// TwinCAT 3 PLC project BE_ObjektH
// ProgramVersion: 3.1.4023.0
// libraries:
//   EfficientIO Communicator, * (EfficientIO)
//   Lynus Energy Basic, * (Lynus AG)
//   Lynus Energy ModbusTCP, * (Lynus AG)
//   Lynus Persistent Data V1, * (Lynus AG)
//   Lynus Standards, * (Lynus AG)
//   Tc2_ModbusSrv, * (Beckhoff Automation GmbH)
//   Tc2_Standard, * (Beckhoff Automation GmbH)
//   Tc2_System, * (Beckhoff Automation GmbH)
//   Tc2_Utilities, * (Beckhoff Automation GmbH)
//   Tc3_IotBase, * (Beckhoff Automation GmbH)
//   Tc3_JsonXml, * (Beckhoff Automation GmbH)
//   Tc3_Module, * (Beckhoff Automation GmbH)
// project tree:
//   / FastTask.TcTTO, MiddleTask.TcTTO, SlowTask.TcTTO (not stored)
//   FB/ FB_ADS_Read.TcPOU, FB_ECS_Keba_P30.TcPOU, FB_Shelly_3EM_not_tested.TcPOU (excluded from build), FB_Shelly_3EM_Helper_not_tested.TcPOU (excluded from build), FB_Shelly_3EM_Helper.TcPOU, FB_Shelly_3EM.TcPOU, F_AdsErrorText.TcPOU
//   POUs/ prgComEffIO.TcPOU, prgCS.TcPOU, prgMain.TcPOU, prgPersistent.TcPOU, prgPV.TcPOU, prgRWEffIO.TcPOU, prgShelly.TcPOU, prgVarEffIO.TcPOU, prg_SystemTime.TcPOU (not stored)
// real-time tasks:
//   TASK FastTask: cycle T#5ms, priority 19, ADS port 350
//   TASK MiddleTask: cycle T#10ms, priority 20, ADS port 351
//   TASK SlowTask: cycle T#20ms, priority 21, ADS port 352

CONFIGURATION BE_ObjektH
    RESOURCE PLC ON TwinCAT3
        TASK FastTask(INTERVAL := T#5ms, PRIORITY := 19);
        TASK MiddleTask(INTERVAL := T#10ms, PRIORITY := 20);
        PROGRAM prgRWEffIO WITH FastTask : prgRWEffIO;
        PROGRAM prgVarEffIO WITH FastTask : prgVarEffIO;
        PROGRAM prg_SystemTime WITH FastTask : prg_SystemTime;
        PROGRAM prgPV WITH MiddleTask : prgPV;
        PROGRAM prgShelly WITH MiddleTask : prgShelly;
        PROGRAM prgCS WITH MiddleTask : prgCS;
        PROGRAM prgPersistent WITH MiddleTask : prgPersistent;
        PROGRAM prgMain WITH MiddleTask : prgMain;
    END_RESOURCE
END_CONFIGURATION

// ---- POUs/prgRWEffIO.TcPOU
PROGRAM prgRWEffIO
VAR
	fbRW1		: FB_ReadWrite_V2;
END_VAR

fbRW1(
	eUploadType:= eSelectDataUploadType.e_Change_Intervall5min , 
	bBusy=> , 
	bError=> , 
	udiErrorCodeOut=> , 
	eErrorReadWrite_Out=> );

END_PROGRAM

// ---- POUs/prgVarEffIO.TcPOU
PROGRAM prgVarEffIO
VAR
	fbVar		: FB_VarInfo;
END_VAR

fbVar(
	bReadInfo:= , 
	eTMCFile:= eSelectTMCFile.eDontUseTMCFile, 
	eSavePositionTMCFile:= eSavePositionOnPLC.ePostionHardDisk, 
	udiCounterFoundVariables=> , 
	bError=> , 
	bBusy=> , 
	byProgress=> , 
	udiErrorCodeOut=> , 
	eErrorVarInfo_Out=> , 
	sVarWithError=> );

END_PROGRAM

// ---- POUs/prgPV.TcPOU
PROGRAM prgPV
VAR
	fbPV					: FB_Symo_PV_Inverter_FLOAT_1_DM_1_Inverter;
	fbPVInt					: FB_PV_Power;
	fbPVCounter				: FB_EnergyCounter;
	lrPowerPV				: LREAL;				//{#lynus.ag#()}
	byErrorWarningPV		: BYTE;					//{#lynus.ag#()}
	bReadyPD_PV				: BOOL;					//{#lynus.ag#()}
	byErrorWarningPD_PV		: BYTE;					//{#lynus.ag#()}
	rHeartbeat_PD_PV		: REAL;					//{#lynus.ag#()}
END_VAR

VAR PERSISTENT
	lrCounterPV				: LREAL;				//{#lynus.ag#()}
END_VAR

fbPV(
	bEnable:= TRUE, 
	sIPAdress:= '192.168.1.3', 
	byUnitID_Inverter:= 1, 
	stDataSymo10=> , 
	stDataEMPower_PV=> , 
	stDataEMCounter_PV=> , 
	diNrOfEM_OUT_PV=> );

fbPVInt(
	bEnable:= TRUE, 
	bPowerDataInvers:= , 
	diNrOfEM_IN_PV:= fbPV.diNrOfEM_OUT_PV, 
	stDataPv=> , 
	diNrOfPv_OUT=> );
	
lrPowerPV := fbPVInt.stDataPv.lrPower;
	byErrorWarningPV := fbPVInt.stDataPv.byErrorWarning;

// EnergyCounter
fbPVCounter(
	byActiveTariff:= 1, 
	lrPowerInput:= 0 - lrPowerPV, 
	lrTotalCounterEnergy_Consumption=> , 
	lrTotalCounterEnergy_Production=> , 
	lrCounterEnergyT1_Consumption=> , 
	lrCounterEnergyT2_Consumption=> , 
	lrCounterEnergyT1_Production=> , 
	lrCounterEnergyT2_Production=> );
	
IF fbPVCounter.lrTotalCounterEnergy_Production > lrCounterPV THEN  	
	lrCounterPV := fbPVCounter.lrTotalCounterEnergy_Production;
END_IF

END_PROGRAM

// ---- POUs/prgShelly.TcPOU
PROGRAM prgShelly
VAR
	// Grid Objekt H 3-phase, 400V
	fbGridObjectH					: FB_Shelly_3EM;
	
	lrPower_ObjectH_Total			: LREAL;			//{#lynus.ag#()}
	lrPower_ObjectH_TotalkW			: LREAL;			//{#lynus.ag#()}
	lrEnergy_ObjectH_Total			: LREAL;			//{#lynus.ag#()}
	lrPower_ObjectH_L1				: LREAL;			//{#lynus.ag#()}
	lrPower_ObjectH_L2				: LREAL;			//{#lynus.ag#()}
	lrPower_ObjectH_L3				: LREAL;			//{#lynus.ag#()}
	lrCurrent_ObjectH_L1			: LREAL;			//{#lynus.ag#()}
	lrCurrent_ObjectH_L2			: LREAL;			//{#lynus.ag#()}
	lrCurrent_ObjectH_L3			: LREAL;			//{#lynus.ag#()}
	lrVoltage_ObjectH_L1			: LREAL;			//{#lynus.ag#()}
	lrVoltage_ObjectH_L2			: LREAL;			//{#lynus.ag#()}
	lrVoltage_ObjectH_L3			: LREAL;			//{#lynus.ag#()}
	lrEnergy_ObjectH_L1				: LREAL;			//{#lynus.ag#()}
	lrEnergy_ObjectH_L2				: LREAL;			//{#lynus.ag#()}
	lrEnergy_ObjectH_L3				: LREAL;			//{#lynus.ag#()}
	
	//21: zuleitung obergeschoss
	
	fbGridSupplyLevel1					: FB_Shelly_3EM;
	
	lrPower_SupplyLevel1_Total			: LREAL;			//{#lynus.ag#()}
	lrPower_SupplyLevel1_TotalkW		: LREAL;			//{#lynus.ag#()}
	lrEnergy_SupplyLevel1_Total			: LREAL;			//{#lynus.ag#()}
	lrPower_SupplyLevel1_L1				: LREAL;			//{#lynus.ag#()}
	lrPower_SupplyLevel1_L2				: LREAL;			//{#lynus.ag#()}
	lrPower_SupplyLevel1_L3				: LREAL;			//{#lynus.ag#()}
	lrCurrent_SupplyLevel1_L1			: LREAL;			//{#lynus.ag#()}
	lrCurrent_SupplyLevel1_L2			: LREAL;			//{#lynus.ag#()}
	lrCurrent_SupplyLevel1_L3			: LREAL;			//{#lynus.ag#()}
	lrVoltage_SupplyLevel1_L1			: LREAL;			//{#lynus.ag#()}
	lrVoltage_SupplyLevel1_L2			: LREAL;			//{#lynus.ag#()}
	lrVoltage_SupplyLevel1_L3			: LREAL;			//{#lynus.ag#()}
	lrEnergy_SupplyLevel1_L1			: LREAL;			//{#lynus.ag#()}
	lrEnergy_SupplyLevel1_L2			: LREAL;			//{#lynus.ag#()}
	lrEnergy_SupplyLevel1_L3			: LREAL;			//{#lynus.ag#()}

	
	//22: Heating
	
	fbGridHeating					: FB_Shelly_3EM;
	
	lrPower_Heating_Total			: LREAL;			//{#lynus.ag#()}
	lrPower_Heating_TotalkW			: LREAL;			//{#lynus.ag#()}
	lrEnergy_Heating_Total			: LREAL;			//{#lynus.ag#()}
	lrPower_Heating_L1				: LREAL;			//{#lynus.ag#()}
	lrPower_Heating_L2				: LREAL;			//{#lynus.ag#()}
	lrPower_Heating_L3				: LREAL;			//{#lynus.ag#()}
	lrCurrent_Heating_L1			: LREAL;			//{#lynus.ag#()}
	lrCurrent_Heating_L2			: LREAL;			//{#lynus.ag#()}
	lrCurrent_Heating_L3			: LREAL;			//{#lynus.ag#()}
	lrVoltage_Heating_L1			: LREAL;			//{#lynus.ag#()}
	lrVoltage_Heating_L2			: LREAL;			//{#lynus.ag#()}
	lrVoltage_Heating_L3			: LREAL;			//{#lynus.ag#()}
	lrEnergy_Heating_L1				: LREAL;			//{#lynus.ag#()}
	lrEnergy_Heating_L2				: LREAL;			//{#lynus.ag#()}
	lrEnergy_Heating_L3				: LREAL;			//{#lynus.ag#()}

	// other
	lrPower_ObjectH_RestkW			: LREAL;			//{#lynus.ag#()}
	lrPower_SupplyLevel1_RestkW		: LREAL;			//{#lynus.ag#()}
	
END_VAR

VAR PERSISTENT
// trigger command execution
	bEnable_GridObjectH				: BOOL:=TRUE;				//{#lynus.ag#()}
	bEnable_SupplyLevel1			: BOOL:=TRUE;				//{#lynus.ag#()}
	bEnable_Heating					: BOOL:=true;				//{#lynus.ag#()}
END_VAR

	// Grid Objekt H 3-phase, 400V
fbGridObjectH(
	bStart:= bEnable_GridObjectH, 
	tDelayRequest:= T#20S, 
	sHostname:= '192.168.0.20', 
	bValidResult=> , 
	bBusy=> , 
	bError=> , 
	bDone=> , 
	hrErrorCode=> ,
	lrtotalpower=> lrPower_ObjectH_Total,
	lrpowerL1=> lrPower_ObjectH_L1,
	lrpowerL2=> lrPower_ObjectH_L2,
	lrpowerL3=> lrPower_ObjectH_L3,
	lrcurrentL1=> lrCurrent_ObjectH_L1,
	lrcurrentL2=> lrCurrent_ObjectH_L2,
	lrcurrentL3=> lrCurrent_ObjectH_L3,
	lrvoltageL1=> lrVoltage_ObjectH_L1,
	lrvoltageL2=> lrVoltage_ObjectH_L2,
	lrvoltageL3=> lrVoltage_ObjectH_L3,
	lrenergyL1=> lrEnergy_ObjectH_L1,
	lrenergyL2=> lrEnergy_ObjectH_L2,
	lrenergyL3=> lrEnergy_ObjectH_L3 );

(* CTs are mounted the wrong way aroung*)	
lrPower_ObjectH_Total	:=	lrPower_ObjectH_Total*(-1);
lrPower_ObjectH_L1		:= 	lrPower_ObjectH_L1*(-1);
lrPower_ObjectH_L2		:= 	lrPower_ObjectH_L2*(-1);
lrPower_ObjectH_L3		:= 	lrPower_ObjectH_L3*(-1);
lrEnergy_ObjectH_L1		:=	lrEnergy_ObjectH_L1*(-1);
lrEnergy_ObjectH_L2		:=	lrEnergy_ObjectH_L2*(-1);
lrEnergy_ObjectH_L3		:=	lrEnergy_ObjectH_L3*(-1);

// re-calc to kW
lrPower_ObjectH_TotalkW := lrPower_ObjectH_Total / 1000;
// sum-up energy
lrEnergy_ObjectH_Total :=  lrEnergy_ObjectH_L1 + lrEnergy_ObjectH_L2 + lrEnergy_ObjectH_L3;

	// Supply Level 1 3-phase, 400V
fbGridSupplyLevel1(
	bStart:= bEnable_SupplyLevel1, 
	tDelayRequest:= T#20S, 
	sHostname:= '192.168.0.21', 
	bValidResult=> , 
	bBusy=> , 
	bError=> , 
	bDone=> , 
	hrErrorCode=> ,
	lrtotalpower=> lrPower_SupplyLevel1_Total,
	lrpowerL1=> lrPower_SupplyLevel1_L1,
	lrpowerL2=> lrPower_SupplyLevel1_L2,
	lrpowerL3=> lrPower_SupplyLevel1_L3,
	lrcurrentL1=> lrCurrent_SupplyLevel1_L1,
	lrcurrentL2=> lrCurrent_SupplyLevel1_L2,
	lrcurrentL3=> lrCurrent_SupplyLevel1_L3,
	lrvoltageL1=> lrVoltage_SupplyLevel1_L1,
	lrvoltageL2=> lrVoltage_SupplyLevel1_L2,
	lrvoltageL3=> lrVoltage_SupplyLevel1_L3,
	lrenergyL1=> lrEnergy_SupplyLevel1_L1,
	lrenergyL2=> lrEnergy_SupplyLevel1_L2,
	lrenergyL3=> lrEnergy_SupplyLevel1_L3 );

(* CTs are mounted the wrong way aroung*)	
lrPower_SupplyLevel1_Total	:=	lrPower_SupplyLevel1_Total*(-1);
lrPower_SupplyLevel1_L1		:= 	lrPower_SupplyLevel1_L1*(-1);
lrPower_SupplyLevel1_L2		:= 	lrPower_SupplyLevel1_L2*(-1);
lrPower_SupplyLevel1_L3		:= 	lrPower_SupplyLevel1_L3*(-1);
lrEnergy_SupplyLevel1_L1		:=	lrEnergy_SupplyLevel1_L1*(-1);
lrEnergy_SupplyLevel1_L2		:=	lrEnergy_SupplyLevel1_L2*(-1);
lrEnergy_SupplyLevel1_L3		:=	lrEnergy_SupplyLevel1_L3*(-1);

// re-calc to kW
lrPower_SupplyLevel1_TotalkW := lrPower_SupplyLevel1_Total / 1000;
// sum-up energy
lrEnergy_SupplyLevel1_Total :=  lrEnergy_SupplyLevel1_L1 + lrEnergy_SupplyLevel1_L2 + lrEnergy_SupplyLevel1_L3;

	// Supply Level 1 3-phase, 400V
fbGridHeating(
	bStart:= bEnable_Heating, 
	tDelayRequest:= T#20S, 
	sHostname:= '192.168.0.22', 
	bValidResult=> , 
	bBusy=> , 
	bError=> , 
	bDone=> , 
	hrErrorCode=> ,
	lrtotalpower=> lrPower_Heating_Total,
	lrpowerL1=> lrPower_Heating_L1,
	lrpowerL2=> lrPower_Heating_L2,
	lrpowerL3=> lrPower_Heating_L3,
	lrcurrentL1=> lrCurrent_Heating_L1,
	lrcurrentL2=> lrCurrent_Heating_L2,
	lrcurrentL3=> lrCurrent_Heating_L3,
	lrvoltageL1=> lrVoltage_Heating_L1,
	lrvoltageL2=> lrVoltage_Heating_L2,
	lrvoltageL3=> lrVoltage_Heating_L3,
	lrenergyL1=> lrEnergy_Heating_L1,
	lrenergyL2=> lrEnergy_Heating_L2,
	lrenergyL3=> lrEnergy_Heating_L3 );

(* CTs are mounted the wrong way aroung*)	
lrPower_Heating_Total	:=	lrPower_Heating_Total*(-1);
lrPower_Heating_L1		:= 	lrPower_Heating_L1*(-1);
lrPower_Heating_L2		:= 	lrPower_Heating_L2*(-1);
lrPower_Heating_L3		:= 	lrPower_Heating_L3*(-1);
lrEnergy_Heating_L1		:=	lrEnergy_Heating_L1*(-1);
lrEnergy_Heating_L2		:=	lrEnergy_Heating_L2*(-1);
lrEnergy_Heating_L3		:=	lrEnergy_Heating_L3*(-1);

// re-calc to kW
lrPower_Heating_TotalkW := lrPower_Heating_Total / 1000;
// sum-up energy
lrEnergy_Heating_Total :=  lrEnergy_Heating_L1 + lrEnergy_Heating_L2 + lrEnergy_Heating_L3;


// other
lrPower_ObjectH_RestkW := lrPower_ObjectH_TotalkW - lrPower_SupplyLevel1_TotalkW;
lrPower_SupplyLevel1_RestkW := lrPower_SupplyLevel1_TotalkW - lrPower_Heating_TotalkW;

END_PROGRAM

// ---- FB/FB_Shelly_3EM.TcPOU
FUNCTION_BLOCK FB_Shelly_3EM
VAR_INPUT
	bStart				: BOOL;
	tDelayRequest		: TIME;		//Timer for delay before start with the next read or write Request
	sHostname			: STRING(255);		//Hostname or IP Adress from the Server
END_VAR

VAR_IN_OUT
END_VAR

VAR_OUTPUT
	bValidResult		: BOOL;							//Valid Result received from Server
    bBusy				: BOOL;							//Function is Busy
    bError				: BOOL;							//Error sucess
	bDone				: BOOL;							//True after the decoding from the received Json File
	bConnected			: BOOL;							//Connection to the Server
	lrtotalpower		: LREAL;						//Received Value
	lrpowerL1			: LREAL;
	lrcurrentL1			: LREAL;
	lrvoltageL1			: LREAL;
	lrenergyL1			: LREAL;
	lrpowerL2			: LREAL;
	lrcurrentL2			: LREAL;
	lrvoltageL2			: LREAL;
	lrenergyL2			: LREAL;
	lrpowerL3			: LREAL;
	lrcurrentL3			: LREAL;
	lrvoltageL3			: LREAL;
	lrenergyL3			: LREAL;
	hrErrorCode       	: HRESULT;						//Error Result from Http Client
END_VAR

VAR
	fbClient			: FB_IotHttpClient;
	fbHttpGet			: FB_Shelly_3EM_Helper;
	timStartRequest		: TON;							//Timer to Start the Request
	FPStartRequest		: R_TRIG;						//Internal positive Edge
	FPDone				: R_TRIG;						//Internal positive Edge
	FNStart				: F_TRIG;						//Internal negative Edge
	y: INT;
END_VAR

(*------------------------------------------------------------------------------------Configure HTTP Client------------------------------------------------------------------------------------------------------*)

fbClient.sHostName := sHostname;
fbClient.tConnectionTimeout := T#30S;

IF NOT fbClient.bConfigured THEN 
	fbClient.nHostPort:= 80;
	fbClient.bKeepAlive := TRUE;
	fbClient.tConnectionTimeout := T#30S;
END_IF


//Timer to start the Request
FPStartRequest(CLK:= bStart, Q=> );
timStartRequest(IN:= fbClient.bConfigured AND bStart AND NOT timStartRequest.Q, PT:= tDelayRequest, Q=> , ET=> );

IF ((timStartRequest.Q AND NOT bBusy) OR (FPStartRequest.Q AND NOT bBusy AND fbClient.bConfigured)) THEN 
	y:=y+1;
	fbHttpGet.bSend := TRUE; 
END_IF

				
//Http Get Function
fbHttpGet(
	lrtotalpower => lrtotalpower, 
	lrpowerL1 => lrpowerL1,
	lrcurrentL1 => lrcurrentL1,
	lrvoltageL1 => lrvoltageL1,
	lrenergyL1 => lrenergyL1,
	lrpowerL2 => lrpowerL2,
	lrcurrentL2 => lrcurrentL2,
	lrvoltageL2 => lrvoltageL2,
	lrenergyL2 => lrenergyL2,
	lrpowerL3 => lrpowerL3,
	lrcurrentL3 => lrcurrentL3,
	lrvoltageL3 => lrvoltageL3,
	lrenergyL3 => lrenergyL3,
	bSend:= , 
	fbClient:= fbClient, 
	bBusy=> bBusy, 
	bError=> ,
	sContentStatus=> ,
	sContentM0=> ,
	sContentM1=> ,
	sContentM2=> );


fbHttpGet.bSend := FALSE;

FPDone(CLK:= bDone, Q=> );

(*
//Http Client
FNStart(CLK:= bStart, Q=> );
	IF FNStart.Q THEN fbClient.Disconnect(); END_IF
*)

fbClient.Execute();

//Error
IF fbHttpGet.bError OR fbClient.bError THEN 
	bError := TRUE; 
ELSE 
	bError := FALSE; 
END_IF	

hrErrorCode := fbClient.hrErrorCode;

END_FUNCTION_BLOCK

// ---- FB/FB_Shelly_3EM_Helper.TcPOU
FUNCTION_BLOCK FB_Shelly_3EM_Helper
VAR_INPUT
	bSend				: BOOL;
END_VAR

VAR_IN_OUT
	fbClient			: FB_IotHttpClient;
END_VAR

VAR_OUTPUT
	bBusy				: BOOL;
	bError				: BOOL;
	lrtotalpower		: LREAL;
	lrpowerL1			: LREAL;
	lrcurrentL1			: LREAL;
	lrvoltageL1			: LREAL;
	lrenergyL1			: LREAL;
	lrpowerL2			: LREAL;
	lrcurrentL2			: LREAL;
	lrvoltageL2			: LREAL;
	lrenergyL2			: LREAL;
	lrpowerL3			: LREAL;
	lrcurrentL3			: LREAL;
	lrvoltageL3			: LREAL;
	lrenergyL3			: LREAL;
END_VAR

VAR
	fbRequestStatus		: FB_IotHttpRequest;
	fbRequestMeter0		: FB_IotHttpRequest;
	fbRequestMeter1		: FB_IotHttpRequest;
	fbRequestMeter2		: FB_IotHttpRequest;
	fbJson				: FB_JsonDomParser;
	nState				: UDINT;
	RisingEdge			: R_TRIG;
	timTimeout			: TON;
	tTimeOut			: TIME := T#50S;
	bGetContentResult	: BOOL;
	sContentStatus		: STRING(511);
	sContentM0			: STRING(511);
	sContentM1			: STRING(511);
	sContentM2			: STRING(511);
	
	bGetJsonResult		: BOOL;
	jsonDoc				: SJsonValue;
	jsonVal				: SJsonValue;
	
	nReqCount			: UDINT;	
	nResCount			: UDINT;
	nValidResCount		: UDINT;
	nErrCount			: UDINT;
	x: INT;
END_VAR

//Timer for Timeout
timTimeout(IN:= nState = 1 AND bBusy, PT:= tTimeOut, Q=> , ET=> );
	IF timTimeout.Q THEN 
		nState := 0;
		bBusy := FALSE;
	END_IF

RisingEdge(CLK:= bSend );
CASE nState OF
0:	
	IF RisingEdge.Q THEN 
		IF 
			fbRequestStatus.SendRequest(sUri:='/status', fbClient:=fbClient, eRequestType:=ETcIotHttpRequestType.HTTP_Get, 0, 0, 0) AND
			fbRequestMeter0.SendRequest(sUri:='/emeter/0', fbClient:=fbClient, eRequestType:=ETcIotHttpRequestType.HTTP_Get, 0, 0, 0) AND 
			fbRequestMeter1.SendRequest(sUri:='/emeter/1', fbClient:=fbClient, eRequestType:=ETcIotHttpRequestType.HTTP_Get, 0, 0, 0) AND
			fbRequestMeter2.SendRequest(sUri:='/emeter/2', fbClient:=fbClient, eRequestType:=ETcIotHttpRequestType.HTTP_Get, 0, 0, 0) THEN				
			nState:= 1;
			nReqCount:= nReqCount+1;
			bBusy:= TRUE;
			bError:= FALSE;
		END_IF					
	END_IF
1:
	x:=x+1;
	IF NOT fbRequestMeter0.bBusy AND NOT fbRequestMeter1.bBusy AND NOT fbRequestMeter2.bBusy AND NOT fbRequestStatus.bBusy THEN
		bError:= TRUE;
		IF NOT fbRequestMeter0.bError THEN				 
			bGetContentResult:= fbRequestMeter0.GetContent(pContent:= ADR(sContentM0), nContentSize:= SIZEOF(sContentM0), bSetNullTermination:= TRUE);
			IF fbRequestMeter0.nStatusCode >= 200 AND fbRequestMeter0.nStatusCode < 300 THEN
				bGetJsonResult:= FALSE;
				jsonDoc:= fbRequestMeter0.GetJsonDomContent(fbJson);
				IF jsonDoc <> 0 THEN
					bGetJsonResult:= TRUE;
					IF fbJson.HasMember(jsonDoc, 'power')  THEN
						jsonVal:= fbJson.FindMember(jsonDoc, 'power');
						nValidResCount:= nValidResCount+1;
						IF fbJson.IsDouble(jsonVal) THEN							
							lrpowerL1:= fbJson.GetDouble(jsonVal);									
						END_IF
						jsonVal:= fbJson.FindMember(jsonDoc, 'current');
						nValidResCount:= nValidResCount+1;
						IF fbJson.IsDouble(jsonVal) THEN							
							lrcurrentL1:= fbJson.GetDouble(jsonVal);									
						END_IF
						jsonVal:= fbJson.FindMember(jsonDoc, 'voltage');
						nValidResCount:= nValidResCount+1;
						IF fbJson.IsDouble(jsonVal) THEN							
							lrvoltageL1:= fbJson.GetDouble(jsonVal);									
						END_IF
						jsonVal:= fbJson.FindMember(jsonDoc, 'total');
						nValidResCount:= nValidResCount+1;
						IF fbJson.IsDouble(jsonVal) THEN							
							lrenergyL1:= fbJson.GetDouble(jsonVal);									
						END_IF	
						bError:= FALSE;
						END_IF
					END_IF						
				nResCount:= nResCount+1;			
				END_IF
		END_IF
		
		IF NOT fbRequestMeter1.bError THEN				 
			bGetContentResult:= fbRequestMeter1.GetContent(pContent:= ADR(sContentM1), nContentSize:= SIZEOF(sContentM1), bSetNullTermination:= TRUE);
			IF fbRequestMeter1.nStatusCode >= 200 AND fbRequestMeter1.nStatusCode < 300 THEN
				bGetJsonResult:= FALSE;
				jsonDoc:= fbRequestMeter1.GetJsonDomContent(fbJson);
				IF jsonDoc <> 0 THEN
					bGetJsonResult:= TRUE;
					IF fbJson.HasMember(jsonDoc, 'power')  THEN
						jsonVal:= fbJson.FindMember(jsonDoc, 'power');
						nValidResCount:= nValidResCount+1;
						IF fbJson.IsDouble(jsonVal) THEN							
							lrpowerL2:= fbJson.GetDouble(jsonVal);									
						END_IF
						jsonVal:= fbJson.FindMember(jsonDoc, 'current');
						nValidResCount:= nValidResCount+1;
						IF fbJson.IsDouble(jsonVal) THEN							
							lrcurrentL2:= fbJson.GetDouble(jsonVal);									
						END_IF
						jsonVal:= fbJson.FindMember(jsonDoc, 'voltage');
						nValidResCount:= nValidResCount+1;
						IF fbJson.IsDouble(jsonVal) THEN							
							lrvoltageL2:= fbJson.GetDouble(jsonVal);									
						END_IF
						jsonVal:= fbJson.FindMember(jsonDoc, 'total');
						nValidResCount:= nValidResCount+1;
						IF fbJson.IsDouble(jsonVal) THEN							
							lrenergyL2:= fbJson.GetDouble(jsonVal);									
						END_IF	
						bError:= FALSE;
						END_IF
					END_IF						
				nResCount:= nResCount+1;			
				END_IF
		END_IF
		
		IF NOT fbRequestMeter2.bError THEN				 
			bGetContentResult:= fbRequestMeter2.GetContent(pContent:= ADR(sContentM2), nContentSize:= SIZEOF(sContentM2), bSetNullTermination:= TRUE);
			IF fbRequestMeter2.nStatusCode >= 200 AND fbRequestMeter2.nStatusCode < 300 THEN
				bGetJsonResult:= FALSE;
				jsonDoc:= fbRequestMeter2.GetJsonDomContent(fbJson);
				IF jsonDoc <> 0 THEN
					bGetJsonResult:= TRUE;
					IF fbJson.HasMember(jsonDoc, 'power')  THEN
						jsonVal:= fbJson.FindMember(jsonDoc, 'power');
						nValidResCount:= nValidResCount+1;
						IF fbJson.IsDouble(jsonVal) THEN							
							lrpowerL3:= fbJson.GetDouble(jsonVal);									
						END_IF
						jsonVal:= fbJson.FindMember(jsonDoc, 'current');
						nValidResCount:= nValidResCount+1;
						IF fbJson.IsDouble(jsonVal) THEN							
							lrcurrentL3:= fbJson.GetDouble(jsonVal);									
						END_IF
						jsonVal:= fbJson.FindMember(jsonDoc, 'voltage');
						nValidResCount:= nValidResCount+1;
						IF fbJson.IsDouble(jsonVal) THEN							
							lrvoltageL3:= fbJson.GetDouble(jsonVal);									
						END_IF
						jsonVal:= fbJson.FindMember(jsonDoc, 'total');
						nValidResCount:= nValidResCount+1;
						IF fbJson.IsDouble(jsonVal) THEN							
							lrenergyL3:= fbJson.GetDouble(jsonVal);									
						END_IF	
						bError:= FALSE;
						END_IF
					END_IF						
				nResCount:= nResCount+1;			
				END_IF
		END_IF
		
		IF NOT fbRequestStatus.bError THEN				 
			bGetContentResult:= fbRequestStatus.GetContent(pContent:= ADR(sContentStatus), nContentSize:= SIZEOF(sContentStatus), bSetNullTermination:= TRUE);
			IF fbRequestStatus.nStatusCode >= 200 AND fbRequestStatus.nStatusCode < 300 THEN
				bGetJsonResult:= FALSE;
				jsonDoc:= fbRequestStatus.GetJsonDomContent(fbJson);
				IF jsonDoc <> 0 THEN
					bGetJsonResult:= TRUE;
					IF fbJson.HasMember(jsonDoc, 'total_power')  THEN
						jsonVal:= fbJson.FindMember(jsonDoc, 'total_power');
						nValidResCount:= nValidResCount+1;
						IF fbJson.IsDouble(jsonVal) THEN							
							lrtotalpower:= fbJson.GetDouble(jsonVal);									
						END_IF
						bError:= FALSE;
					END_IF
				END_IF		
				nResCount:= nResCount+1;			
			END_IF
		END_IF
		
		nState:= 0;
		bBusy:= FALSE;
		IF bError THEN
			nErrCount:= nErrCount+1;
		END_IF
	END_IF  	
END_CASE

END_FUNCTION_BLOCK

// ---- POUs/prgCS.TcPOU
PROGRAM prgCS
VAR
	fbCS1	:	FB_ECS_Keba_P30;
	bEnableCS1	: BOOL:=TRUE;
	
	lr_CS1_TotalPower_KebaP30: LREAL;						//{#lynus.ag#()}
	b_CS1_CarConnected: BOOL;								//{#lynus.ag#()}
	i_CS1_CarConnectedInd: INT;								//{#lynus.ag#()}
	b_CS1_Enabled: BOOL;									//{#lynus.ag#()}
	b_CS1_OutputOn: BOOL;									//{#lynus.ag#()}
	dw_CS1_ChargingState: DWORD;							//{#lynus.ag#()}
	dw_CS1_ErrorCode: DWORD;								//{#lynus.ag#()}
	lreal_CS1_TotalEnergyConsumption: LREAL;				//{#lynus.ag#()}
	lreal_CS1_EnergySession: LREAL;							//{#lynus.ag#()}
	lreal_CS1_Serial: LREAL;								//{#lynus.ag#()}

	fbCS2	:	FB_ECS_Keba_P30;
	bEnableCS2	: BOOL:=TRUE;
	
	lr_CS2_TotalPower_KebaP30: LREAL;						//{#lynus.ag#()}
	b_CS2_CarConnected: BOOL;								//{#lynus.ag#()}
	i_CS2_CarConnectedInd: INT;								//{#lynus.ag#()}
	b_CS2_Enabled: BOOL;									//{#lynus.ag#()}
	b_CS2_OutputOn: BOOL;									//{#lynus.ag#()}
	dw_CS2_ChargingState: DWORD;							//{#lynus.ag#()}
	dw_CS2_ErrorCode: DWORD;								//{#lynus.ag#()}
	lreal_CS2_TotalEnergyConsumption: LREAL;				//{#lynus.ag#()}
	lreal_CS2_EnergySession: LREAL;							//{#lynus.ag#()}
	lreal_CS2_Serial: LREAL;								//{#lynus.ag#()}

	fbCS3	:	FB_ECS_Keba_P30;
	bEnableCS3	: BOOL:=TRUE;
	
	lr_CS3_TotalPower_KebaP30: LREAL;						//{#lynus.ag#()}
	b_CS3_CarConnected: BOOL;								//{#lynus.ag#()}
	i_CS3_CarConnectedInd: INT;								//{#lynus.ag#()}
	b_CS3_Enabled: BOOL;									//{#lynus.ag#()}
	b_CS3_OutputOn: BOOL;									//{#lynus.ag#()}
	dw_CS3_ChargingState: DWORD;							//{#lynus.ag#()}
	dw_CS3_ErrorCode: DWORD;								//{#lynus.ag#()}
	lreal_CS3_TotalEnergyConsumption: LREAL;				//{#lynus.ag#()}
	lreal_CS3_EnergySession: LREAL;							//{#lynus.ag#()}
	lreal_CS3_Serial: LREAL;								//{#lynus.ag#()}

	r_trig_Errror	:r_trig;
	iCount: INT;
	Str_IP: STRING(25);
	i_ErrorCount: INT;
	Str_IP_1: STRING(25):= '192.168.0.113';
	Str_IP_2: STRING(25):= '192.168.0.114';
	Str_IP_3: STRING(25):= '192.168.0.115';

END_VAR
VAR PERSISTENT
END_VAR

fbCS1(
	bEnable:= bEnableCS1, 
	bPowerDataInvers:=TRUE , 
	byElectricFuseLine:= ,
	uiFailsafeCurrent:=32000,
	uiFailsafeTimeOut:=600,
	diNrOfEMS_IN:= , 
	diNrOfEM_IN_CS:= , 
	sIPAdress:= Str_IP_1,			// .113 = Seriennummer 17211656
	stSetupECS:= , 
	stDataECS=> , 
	diNrOfECS_OUT=> , 
	lrTotalPowerECSRealTime=> );
	
	
	lr_CS1_TotalPower_KebaP30 			:=	fbCS1.lrTotalPowerECSRealTime;
	b_CS1_CarConnected				 	:=	fbCS1.stDataECS.bCarConnected;
	b_CS1_Enabled						:= 	fbCS1.stDataECS.bEnabled;
	b_CS1_OutputOn						:=	fbCS1.stDataECS.bOutputOnOff;
	dw_CS1_ChargingState				:=  fbCs1.dwChargingState;
	dw_CS1_ErrorCode					:=  fbCs1.dwErrorCode;
	lreal_CS1_TotalEnergyConsumption	:=	fbCS1.lrTotalCounterEnergy_Consumption/1000;
	lreal_CS1_EnergySession				:=	fbCS1.lrChargedEnergySession;
	lreal_CS1_Serial					:=  fbCS1.lr_Serial;
	
	IF b_CS1_CarConnected = TRUE THEN
		i_CS1_CarConnectedInd := 251;
		ELSE i_CS1_CarConnectedInd := 0;
	END_IF

	(*
// zum probieren der IP

// scan Modbus IP address

r_trig_Errror(CLK:=fbCS1.fbMBRead_FC3.bError);

IF r_trig_Errror.Q THEN
	i_ErrorCount := i_ErrorCount+1;
	IF i_ErrorCount>10 THEN 
		i_ErrorCount:=0;
		iCount:=iCount+1;
		IF iCount <0 OR iCount >255 THEN
			iCount := 1;
		END_IF
	ELSE
		i_ErrorCount:=i_ErrorCount+1;
	END_IF
END_IF	

Str_IP := concat('192.168.42.',INT_TO_STRING(iCount));
*)	
	
	
fbCS2(
	bEnable:= bEnableCS2, 
	bPowerDataInvers:=TRUE , 
	byElectricFuseLine:= ,
	uiFailsafeCurrent:=32000,
	uiFailsafeTimeOut:=600,
	diNrOfEMS_IN:= , 
	diNrOfEM_IN_CS:= , 
	sIPAdress:= Str_IP_2, 				// .114 = Seriennummer 17111777
	stSetupECS:= , 
	stDataECS=> , 
	diNrOfECS_OUT=> , 
	lrTotalPowerECSRealTime=> );
	
	
	lr_CS2_TotalPower_KebaP30 			:=	fbCS2.lrTotalPowerECSRealTime;
	b_CS2_CarConnected				 	:=	fbCS2.stDataECS.bCarConnected;
	b_CS2_Enabled						:= 	fbCS2.stDataECS.bEnabled;
	b_CS2_OutputOn						:=	fbCS2.stDataECS.bOutputOnOff;
	dw_CS2_ChargingState				:=  fbCS2.dwChargingState;
	dw_CS2_ErrorCode					:=  fbCS2.dwErrorCode;
	lreal_CS2_TotalEnergyConsumption	:=	fbCS2.lrTotalCounterEnergy_Consumption/1000;
	lreal_CS2_EnergySession				:=	fbCS2.lrChargedEnergySession;
	lreal_CS2_Serial					:=  fbCS2.lr_Serial;
	
	IF b_CS2_CarConnected = TRUE THEN
		i_CS2_CarConnectedInd := 251;
		ELSE i_CS2_CarConnectedInd := 0;
	END_IF
	
fbCS3(
	bEnable:= bEnableCS3, 
	bPowerDataInvers:=TRUE , 
	byElectricFuseLine:= ,
	uiFailsafeCurrent:=32000,
	uiFailsafeTimeOut:=600,
	diNrOfEMS_IN:= , 
	diNrOfEM_IN_CS:= , 
	sIPAdress:= Str_IP_3, 			// .115 = Seriennummer 19326220
	stSetupECS:= , 
	stDataECS=> , 
	diNrOfECS_OUT=> , 
	lrTotalPowerECSRealTime=> );
	
	
	lr_CS3_TotalPower_KebaP30 			:=	fbCS3.lrTotalPowerECSRealTime;
	b_CS3_CarConnected				 	:=	fbCS3.stDataECS.bCarConnected;
	b_CS3_Enabled						:= 	fbCS3.stDataECS.bEnabled;
	b_CS3_OutputOn						:=	fbCS3.stDataECS.bOutputOnOff;
	dw_CS3_ChargingState				:=  fbCS3.dwChargingState;
	dw_CS3_ErrorCode					:=  fbCS3.dwErrorCode;
	lreal_CS3_TotalEnergyConsumption	:=	fbCS3.lrTotalCounterEnergy_Consumption/1000;
	lreal_CS3_EnergySession				:=	fbCS3.lrChargedEnergySession;
	lreal_CS3_Serial					:=  fbCS3.lr_Serial;
	
	IF b_CS3_CarConnected = TRUE THEN
		i_CS3_CarConnectedInd := 251;
		ELSE i_CS3_CarConnectedInd := 0;
	END_IF

END_PROGRAM

// ---- FB/FB_ECS_Keba_P30.TcPOU
FUNCTION_BLOCK FB_ECS_Keba_P30
VAR_INPUT PERSISTENT
	///{#lynus.ag#()} //Enable the Fuctionblock and his logic
	bEnable: BOOL;
	///With True its possible to invert all received power data from the electric meter
	bPowerDataInvers: BOOL;
	///Electric Fuse Line on wich the ECS is connected => 1 2 3 (If 0 then this charging station is not connected to a Electric Fuse Line)
	byElectricFuseLine: BYTE;
	///Failsafe Current when the connection between PLC and Charging station is interrupted. 0mA = CS Off, 6000mA - 32000mA
	uiFailsafeCurrent: UINT;
	///Failsafe Timeout when the connection between PLC and Charging station is interrupted. 10 - 600 sec
	uiFailsafeTimeOut: UINT := 10;
	///Number of EMS what control this Device.
	diNrOfEMS_IN: DINT;
	///Number of the electric meter for incoming power data. (Power Data for this Device)
	diNrOfEM_IN_CS: DINT;
	///IP Adress from the Keba charging station
	sIPAdress: STRING(15);
	///{#lynus.ag#()} //Setup charging station
	stSetupECS: ST_Setup_ECS;
END_VAR
VAR_OUTPUT
	///{#lynus.ag#()} //Electric charging station output data
	stDataECS: ST_ECS_Output;
	///Active Number from the Electric charging Function for using on other functions
	diNrOfECS_OUT: DINT;
	///Total Electric Power in kW read out directly from the Charging station. (Real time)
	lrTotalPowerECSRealTime: LREAL; 

	lr_Serial: LREAL;		
END_VAR
VAR
	///Function block for electric charging station
	
	fbCS: FB_ElectricChargingStation;
	///Function block to calcualte the number of the Device
	
	fbNumberDevice: FB_NumberOfDevice;
	///Digital Input from external loock signal
	fbDIExternalLock: FB_XL1XXX_DI;
	///Modbus Read Function (FC3)
	
	fbMBRead_FC3: FB_MBReadRegs;
	///Modbus Write Function (FC6)
	
	fbMBWrite_FC6: FB_MBWriteSingleReg;
	///Convert Word to Dword
	
	fbConvertWordToDword: FB_CV_WORD_TO_DWORD;
	///Timer for Delay between Requests
	
	timDelay: TON;
	///Timer for Timeout
	
	timTimeout: TON;
	///Timer to dissable the Function after Lynus_Standards.Constants_General.tTimeDissableLynusFunctions Days without connection to the Lynus Cloud
	
	timDissableFunctions: TON;
	///Timer to try reset the connection Flag on the GVL. (When somebody delete the Connection Function and make only a onlinechange)
	
	timResetConnectionOnGVL: TON;
	///Charging Time
	
	timChTimeSocket: TON;
	///Timer to start the state machine with Daley after enabling or after the system ist restartet
	
	timDelayStart: TON;
	///Timer to Close the Socket after to much Errors
	
	timCloseSocket: TON;
	///Internal positive Edge
	
	FPError_FC_3: R_TRIG;
	///Internal positive Edge
	
	FPError_FC_6: R_TRIG;
	///Internal positive Edge
	
	FPEnable: R_TRIG;
	///Function to save persistent data
	
	arrPD: ARRAY[1..16] OF FB_PersistentData_Number;
	///Function to save persistent string data
	
	fbPDString: FB_PersistentData_String;
	///Buffer with Data from FC3
	
	arrBuffer_FC3: ARRAY[1..2] OF WORD;
	///Error State from the charging station
	
	bErrorCS: BOOL;
	///Modbus TCP Function Error Counter																	
	
	byMBTCPErrorCounter: BYTE;
	///Wait in Step before start to clean data on PLC
	
	byWaitInStep: BYTE;
	///State machine to handle the data on the GVL
	
	iStateGVLData: INT;
	///State machine for read out Data over Modbus TCP
	
	iStateModbusRead: INT;
	///State machine for write Data over Modbus TCP
	
	iStateModbusWrite: INT;
	///State machine for error out Data over Modbus TCP	
	
	iStateModbusError: INT;
	///Variable to compare the state machine variable to set or reset the timeout timer
	
	iStateModbus_CP: INT;
	///Number of active batterys
	
	diNumberOfActiveBatterys: DINT;
	///Number of battery inverters that work in Emergency Power operation 
	
	diNumberOfBatteryInverterInEPO: DINT;
	///Loop to clean old data on GVL
	
	diLPForGVL: DINT;
	///Counter to clean old data on GVL
	
	diCounterForGVL: DINT;
	///Sum of the SOC from all batterys
	
	dwSumSOC: DWORD;
	///Charging State from the Keba Charger
	
	dwChargingState: DWORD;
	///Cable State from the Keba Charger
	
	dwCableState: DWORD;
	///Error Code from the Keba Charger
	
	dwErrorCode: DWORD;
	///Power from the ECS in W 
	
	rPowerECS: REAL;
	///Energy Counter Consumption in Wh
	
	lrTotalCounterEnergy_Consumption: LREAL;
	///Charged Energy from the active Session in Wh
	
	lrChargedEnergySession: LREAL;
	///Loop to check some data from batterys
	
	liLPBatteryData: LINT;
	///Loop to check if 1 or more battery inverters build a island grid
	
	liLPInEPO: LINT;
	i: INT;
	word_MBadress: WORD;

END_VAR
VAR PERSISTENT
	///Number of EMS what control this Device to compare with the original
	{attribute 'conditionalshow' := ''}
	diNrOfEMS_IN_CP: DINT;
END_VAR

//Creator : Kai Ebensperger
//Company : Lynus AG
//Date : 15.07.2022
//Version : 1.0.0.0

//With this Funcition its possible to communicate with a Keba P30 Charging station over Modbus TCP.
//Support the C-Series from Version 3.10.16 or higher
//Support the X-Series from Version 1.11 or higher
//Its possible to controll the charging station over the charge current
//When the Function send 0 Ampere is switched of, then the charging station is blocked and its not possible to charge
//The Communication is not so fast because in the Documentation they write that we can read every 500MS but we can write onle ever 5 seconds.
//We can read only 1 Register at each command. Its not possible to read more Registers with 1 command
//The Unit ID is always 255
//Also the Settings for Fail Save is includes in ths Fuction. The Failsave Current is set to uiFailsafeCurrent.
//Failsafe takes effect when the connection between the PLC and the charging station is interrupted. Timout is uiFailsafeTimeOut in seconds.

//Versions that are supported : 1.3

//NOTE for diNr.....Designation => 
//_IN = Here Data come in from other Functions or go out to other functions about the GVL
//_OUT = Here Data go out to other functions about the GVL

(*--------------------------------------------------------------------------------------------Limits-------------------------------------------------------------------------------------*)

diNrOfEMS_IN := LIMIT(0,diNrOfEMS_IN,Constants_Energy.diMaxNumberOfEMS);
	diNrOfEM_IN_CS := LIMIT(0,diNrOfEM_IN_CS,Constants_Energy.diMaxNumberOfElectricMeters);
		byElectricFuseLine := LIMIT(0,byElectricFuseLine,30);
			IF uiFailsafeCurrent > 0 THEN 
				uiFailsafeCurrent := LIMIT(6000,uiFailsafeCurrent,32000);
			END_IF 
				uiFailsafeTimeOut := LIMIT(10,uiFailsafeTimeOut,600);	
		
(*------------------------------------------------------------------Power Data----------------------------------------------------------------------------*)

IF diNrOfEM_IN_CS <> 0 THEN
	//Energy Session Input data
	fbCS.bCalculateEnergySession := FALSE;
	fbCS.arrSocketPowerECS[1] := 0;
	fbCS.arrSocketPowerECS[2] := 0;
	fbCS.arrSocketPowerECS[3] := 0;
	fbCS.arrSocketPowerECS[4] := 0;
	fbCS.arrSocketEnergySession[1] := 0;
	fbCS.arrSocketEnergySession[2] := 0;
	fbCS.arrSocketEnergySession[3] := 0;
	fbCS.arrSocketEnergySession[4] := 0;
		IF NOT bPowerDataInvers THEN
			//Energy meter input data for cs Function block
			fbCS.lrCounterEnergyT1_Consumption := Lynus_Standards.GVL_Energy.stDataElectricMeters[diNrOfEM_IN_CS].lrCounterEnergyT1_Production * 1000;
			fbCS.lrCounterEnergyT2_Consumption := Lynus_Standards.GVL_Energy.stDataElectricMeters[diNrOfEM_IN_CS].lrCounterEnergyT2_Production * 1000;
			fbCS.lrCounterEnergyT1_Production := Lynus_Standards.GVL_Energy.stDataElectricMeters[diNrOfEM_IN_CS].lrCounterEnergyT1_Consumption * 1000;
			fbCS.lrCounterEnergyT2_Production := Lynus_Standards.GVL_Energy.stDataElectricMeters[diNrOfEM_IN_CS].lrCounterEnergyT1_Consumption * 1000;
			fbCS.lrTotalCounterEnergy_Consumption := Lynus_Standards.GVL_Energy.stDataElectricMeters[diNrOfEM_IN_CS].lrTotalCounterEnergy_Production * 1000;
			fbCS.lrTotalCounterEnergy_Production := Lynus_Standards.GVL_Energy.stDataElectricMeters[diNrOfEM_IN_CS].lrTotalCounterEnergy_Consumption * 1000;
				fbCS.lrTotalPowerECS := (Lynus_Standards.GVL_Energy.stDataElectricMeters[diNrOfEM_IN_CS].lrPower * 1000) * -1;
			ELSE
			//Energy meter input data for cs Function block
			fbCS.lrCounterEnergyT1_Consumption := Lynus_Standards.GVL_Energy.stDataElectricMeters[diNrOfEM_IN_CS].lrCounterEnergyT1_Consumption * 1000;
			fbCS.lrCounterEnergyT2_Consumption := Lynus_Standards.GVL_Energy.stDataElectricMeters[diNrOfEM_IN_CS].lrCounterEnergyT2_Consumption * 1000;
			fbCS.lrCounterEnergyT1_Production := Lynus_Standards.GVL_Energy.stDataElectricMeters[diNrOfEM_IN_CS].lrCounterEnergyT1_Production * 1000;
			fbCS.lrCounterEnergyT2_Production := Lynus_Standards.GVL_Energy.stDataElectricMeters[diNrOfEM_IN_CS].lrCounterEnergyT2_Production * 1000;
			fbCS.lrTotalCounterEnergy_Consumption := Lynus_Standards.GVL_Energy.stDataElectricMeters[diNrOfEM_IN_CS].lrTotalCounterEnergy_Consumption * 1000;
			fbCS.lrTotalCounterEnergy_Production := Lynus_Standards.GVL_Energy.stDataElectricMeters[diNrOfEM_IN_CS].lrTotalCounterEnergy_Production * 1000;
				fbCS.lrTotalPowerECS := Lynus_Standards.GVL_Energy.stDataElectricMeters[diNrOfEM_IN_CS].lrPower * 1000;
		END_IF
ELSE
	//Energy meter input data for cs Function block
	fbCS.lrCounterEnergyT1_Consumption := lrTotalCounterEnergy_Consumption;
	fbCS.lrCounterEnergyT2_Consumption := 0;
	fbCS.lrCounterEnergyT1_Production := 0;
	fbCS.lrCounterEnergyT2_Production := 0;
	fbCS.lrTotalCounterEnergy_Consumption := lrTotalCounterEnergy_Consumption;
	fbCS.lrTotalCounterEnergy_Production := 0;
		fbCS.lrTotalPowerECS := rPowerECS;
	//Energy Session Input data
	fbCS.bCalculateEnergySession := FALSE;
	fbCS.arrSocketPowerECS[1] := rPowerECS;
	fbCS.arrSocketPowerECS[2] := 0;
	fbCS.arrSocketPowerECS[3] := 0;
	fbCS.arrSocketPowerECS[4] := 0;
	fbCS.arrSocketEnergySession[1] := lrChargedEnergySession;
	fbCS.arrSocketEnergySession[2] := 0;
	fbCS.arrSocketEnergySession[3] := 0;
	fbCS.arrSocketEnergySession[4] := 0;
END_IF			

(*-------------------------------------------------------------Calcualte the number of ECS---------------------------------------------------------------*)

fbNumberDevice(
	diActualNumberOfDevices:= Lynus_Standards.GVL_Energy.stNumberOfDevices.diNumberOfECS, 
	diMaxNumberOfDevices:= Constants_Energy.diMaxNumberOfElectricChargingStations, 
	udiCounterOnlineChange:= TwinCAT_SystemInfoVarList._AppInfo.OnlineChangeCnt, 
	bNumberIsCalculatet=> , 
	bFPNumberIsCalculatet=> , 
	bOnlineChange=> , 
	diNumberForThisDevice=> diNrOfECS_OUT, 
	diNumberOfTotalDevices=> );

//Write new Numer on GVL
IF fbNumberDevice.bFPNumberIsCalculatet THEN
	Lynus_Standards.GVL_Energy.stNumberOfDevices.diNumberOfECS := fbNumberDevice.diNumberOfTotalDevices;	
END_IF 

//Delete old Number on GVL
IF fbNumberDevice.bOnlineChange THEN 
	Lynus_Standards.GVL_Energy.stNumberOfDevices.diNumberOfECS := diNrOfECS_OUT;	
		iStateGVLData := 1;
END_IF

(*-------------------------------------------------------------Service from Backend is ready and check the connection to backen for dissabel/enable Function---------------------------------------------------------------*)

//Try to reset the variable for connection on the GVL. When all is normal then the Lynus Mqtt connection function set this variable to true in the next cycle
//When we have no connection to the backend then after Lynus_Standards.Constants_General.tTimeDissableLynusFunctions days the Function is dissabled with all of his functionalities
timResetConnectionOnGVL(IN:= NOT timResetConnectionOnGVL.Q, PT:= T#1H, Q=> , ET=> );
	IF timResetConnectionOnGVL.Q THEN Lynus_Standards.GVL_Communicator.bStateConnectionToEnableFunctions := FALSE; END_IF
		IF NOT Lynus_Standards.GVL_Communicator.bStateConnectionToEnableFunctions THEN timDissableFunctions.IN := TRUE; ELSE timDissableFunctions.IN := FALSE; END_IF  
			timDissableFunctions(IN:= , PT:= Lynus_Standards.Constants_General.tTimeDissableLynusFunctions, Q=> , ET=> );
			
(*--------------------------------------------------------------------------------------------State Machine Read--------------------------------------------------------------------------------------*)

//Timer for Delay
timDelay(IN:= , PT:= T#750MS, Q=> , ET=> );

//Timer for Timeout in Statemachine
IF (iStateModbusRead > 0 AND iStateModbusRead <= 7 AND iStateModbusRead = iStateModbus_CP) OR
		(iStateModbusWrite > 0 AND iStateModbusWrite <= 2 AND iStateModbusWrite = iStateModbus_CP) THEN
			timTimeout.IN := TRUE;
ELSE	
			timTimeout.IN := FALSE;
END_IF
	//Timeout Timer is dissabled when the Init Step is aktiv or the function is not enabled
	IF (iStateModbusRead = 0 AND iStateModbusWrite = 0) OR NOT bEnable THEN timTimeout.IN := FALSE; END_IF
		timTimeout(IN:= , PT:= T#10S, Q=> , ET=> );

//Enable with Delay that not all sockets have to be created at the same time
timDelayStart(IN:= bEnable, PT:= T#20MS * diNrOfECS_OUT, Q=> , ET=> );
	FPEnable(CLK:= timDelayStart.Q, Q=> );

IF FPEnable.Q AND iStateModbusRead = 0 AND iStateModbusWrite = 0 THEN iStateModbusRead := 1; END_IF		
		
//Not Enabled
IF NOT bEnable THEN iStateModbusRead := 0; iStateModbusError := 0; iStateModbusWrite := 0; END_IF		
		
CASE iStateModbusRead OF
	 
	0://Init Step 
		iStateModbus_CP := 0;
			timDelay.IN := FALSE;
				fbMBRead_FC3.bExecute := FALSE;
					fbMBWrite_FC6.bExecute := FALSE;
						rPowerECS := 0;
							dwChargingState := 0;
								dwCableState := 0;	
									lrChargedEnergySession := 0;
	
	1://Charging State (Register 1000) !!!!Maybe 0 or 1....test it. Then change also the other Register Adresses!!!!!
		iStateModbus_CP := iStateModbusRead;

		//Start Read
		fbMBRead_FC3.nQuantity := 2;
			fbMBRead_FC3.nMBAddr := 1000;
				fbMBRead_FC3.bExecute := TRUE;
					fbMBRead_FC3.nUnitID := 255;
			
		IF fbMBRead_FC3.bBusy THEN timDelay.IN := TRUE; END_IF
		
		//Wait for Delay, copy Data and then next step
		IF NOT fbMBRead_FC3.bBusy AND NOT fbMBRead_FC3.bError AND timDelay.Q THEN
			//Charging State
			fbConvertWordToDword(wInputValue_1:= arrBuffer_FC3[1], wInputValue_2:= arrBuffer_FC3[2], eByteOrderForConvert:= eByteOrder.eBigEndian, dwOutputValue =>);
				dwChargingState := fbConvertWordToDword.dwOutputValue;
			
			//Go to Next Step
			fbMBRead_FC3.bExecute := FALSE;
				timDelay.IN := FALSE;		
					iStateModbusRead := 2;
		END_IF	

		//Error or Timeout
		IF FPError_FC_3.Q OR timTimeout.Q THEN
			iStateModbusError := 300;
		END_IF	
		
	2://Cable State (Register 1004)
		iStateModbus_CP := iStateModbusRead;

		//Start Read
		fbMBRead_FC3.nQuantity := 2;
			fbMBRead_FC3.nMBAddr := 1004;
				fbMBRead_FC3.bExecute := TRUE;
					fbMBRead_FC3.nUnitID := 255;
			
		IF fbMBRead_FC3.bBusy THEN timDelay.IN := TRUE; END_IF
		
		//Wait for Delay, copy Data and then next step
		IF NOT fbMBRead_FC3.bBusy AND NOT fbMBRead_FC3.bError AND timDelay.Q THEN
			//Cable State
			fbConvertWordToDword(wInputValue_1:= arrBuffer_FC3[1], wInputValue_2:= arrBuffer_FC3[2], eByteOrderForConvert:= eByteOrder.eBigEndian, dwOutputValue =>);
				dwCableState := fbConvertWordToDword.dwOutputValue;
			//Go to Next Step
			fbMBRead_FC3.bExecute := FALSE;
				timDelay.IN := FALSE;		
					iStateModbusRead := 3;
		END_IF	

		//Error or Timeout
		IF FPError_FC_3.Q OR timTimeout.Q THEN
			iStateModbusError := 300;
		END_IF	
		
	3://Error Code (Register 1006)
		iStateModbus_CP := iStateModbusRead;

		//Start Read
		fbMBRead_FC3.nQuantity := 2;
			fbMBRead_FC3.nMBAddr := 1006;
				fbMBRead_FC3.bExecute := TRUE;
					fbMBRead_FC3.nUnitID := 255;
			
		IF fbMBRead_FC3.bBusy THEN timDelay.IN := TRUE; END_IF
		
		//Wait for Delay, copy Data and then next step
		IF NOT fbMBRead_FC3.bBusy AND NOT fbMBRead_FC3.bError AND timDelay.Q THEN
			//Error Code
			fbConvertWordToDword(wInputValue_1:= arrBuffer_FC3[1], wInputValue_2:= arrBuffer_FC3[2], eByteOrderForConvert:= eByteOrder.eBigEndian, dwOutputValue =>);
				dwErrorCode := fbConvertWordToDword.dwOutputValue;
			//Go to Next Step
			fbMBRead_FC3.bExecute := FALSE;
				timDelay.IN := FALSE;		
					iStateModbusRead := 4;
		END_IF	

		//Error or Timeout
		IF FPError_FC_3.Q OR timTimeout.Q THEN
			iStateModbusError := 300;
		END_IF	
		
	4://Active Power (Register 1020)
		iStateModbus_CP := iStateModbusRead;

		//Start Read
		fbMBRead_FC3.nQuantity := 2;
			fbMBRead_FC3.nMBAddr := 1020;
				fbMBRead_FC3.bExecute := TRUE;
					fbMBRead_FC3.nUnitID := 255;
			
		IF fbMBRead_FC3.bBusy THEN timDelay.IN := TRUE; END_IF
		
		//Wait for Delay, copy Data and then next step
		IF NOT fbMBRead_FC3.bBusy AND NOT fbMBRead_FC3.bError AND timDelay.Q THEN
			//Active Power in mW
			fbConvertWordToDword(wInputValue_1:= arrBuffer_FC3[1], wInputValue_2:= arrBuffer_FC3[2], eByteOrderForConvert:= eByteOrder.eBigEndian, dwOutputValue =>);
				rPowerECS := DWORD_TO_REAL(fbConvertWordToDword.dwOutputValue);
					rPowerECS := rPowerECS / 1000;	
			//Go to Next Step
			fbMBRead_FC3.bExecute := FALSE;
				timDelay.IN := FALSE;		
					iStateModbusRead := 5;
		END_IF	

		//Error or Timeout
		IF FPError_FC_3.Q OR timTimeout.Q THEN
			iStateModbusError := 300;
		END_IF	
	
	5://Total Energy (Register 1036)
		iStateModbus_CP := iStateModbusRead;

		//Start Read
		fbMBRead_FC3.nQuantity := 2;
			fbMBRead_FC3.nMBAddr := 1036;
				fbMBRead_FC3.bExecute := TRUE;
					fbMBRead_FC3.nUnitID := 255;
			
		IF fbMBRead_FC3.bBusy THEN timDelay.IN := TRUE; END_IF
		
		//Wait for Delay, copy Data and then next step
		IF NOT fbMBRead_FC3.bBusy AND NOT fbMBRead_FC3.bError AND timDelay.Q THEN
			//Total Energy in Wh
			fbConvertWordToDword(wInputValue_1:= arrBuffer_FC3[1], wInputValue_2:= arrBuffer_FC3[2], eByteOrderForConvert:= eByteOrder.eBigEndian, dwOutputValue =>);
				lrTotalCounterEnergy_Consumption := DWORD_TO_LREAL(fbConvertWordToDword.dwOutputValue);
			//Go to Next Step
			fbMBRead_FC3.bExecute := FALSE;
				timDelay.IN := FALSE;		
					iStateModbusRead := 6;
		END_IF	

		//Error or Timeout
		IF FPError_FC_3.Q OR timTimeout.Q THEN
			iStateModbusError := 300;
		END_IF	
		
	6://Charged Energy from current charging session (Register 1502)
		iStateModbus_CP := iStateModbusRead;

		//Start Read
		fbMBRead_FC3.nQuantity := 2;
			fbMBRead_FC3.nMBAddr := 1502;
				fbMBRead_FC3.bExecute := TRUE;
					fbMBRead_FC3.nUnitID := 255;
			
		IF fbMBRead_FC3.bBusy THEN timDelay.IN := TRUE; END_IF
		
		//Wait for Delay, copy Data and then next step
		IF NOT fbMBRead_FC3.bBusy AND NOT fbMBRead_FC3.bError AND timDelay.Q THEN
			//Total Energy in Wh
			fbConvertWordToDword(wInputValue_1:= arrBuffer_FC3[1], wInputValue_2:= arrBuffer_FC3[2], eByteOrderForConvert:= eByteOrder.eBigEndian, dwOutputValue =>);
				lrChargedEnergySession := DWORD_TO_LREAL(fbConvertWordToDword.dwOutputValue);
			//Go to Next Step
			fbMBRead_FC3.bExecute := FALSE;
				timDelay.IN := FALSE;		
					iStateModbusRead := 7;
		END_IF	

		//Error or Timeout
		IF FPError_FC_3.Q OR timTimeout.Q THEN
			iStateModbusError := 300;
		END_IF	
		
	7://Serial number (Register 1014)
		iStateModbus_CP := iStateModbusRead;

		//Start Read
		fbMBRead_FC3.nQuantity := 2;
		fbMBRead_FC3.nMBAddr := 1014;
		fbMBRead_FC3.bExecute := TRUE;
		fbMBRead_FC3.nUnitID := 255;
			
		IF fbMBRead_FC3.bBusy THEN timDelay.IN := TRUE; END_IF
		
		//Wait for Delay, copy Data and then next step
		IF NOT fbMBRead_FC3.bBusy AND NOT fbMBRead_FC3.bError AND timDelay.Q THEN
			//Total Energy in Wh
			fbConvertWordToDword(wInputValue_1:= arrBuffer_FC3[1], wInputValue_2:= arrBuffer_FC3[2], eByteOrderForConvert:= eByteOrder.eBigEndian, dwOutputValue =>);
			lr_Serial := DWORD_TO_LREAL(fbConvertWordToDword.dwOutputValue);
			//Go to Next Step
			fbMBRead_FC3.bExecute := FALSE;
			timDelay.IN := FALSE;		
			iStateModbusRead := 8;
		END_IF	

		//Error or Timeout
		IF FPError_FC_3.Q OR timTimeout.Q THEN
			iStateModbusError := 300;
		END_IF	

	8://Wait 1 Step to reset the delay counter befor start to write
		iStateModbus_CP := iStateModbusRead;
		
			// iStateModbusWrite := 1;
				//-1 because 0 is the Init Step for Read
			//	iStateModbusRead := -1;   
				iStateModbusRead := 1;   
				
			//Error on Master, changes on Inputs or Timeout
		 	IF timTimeout.Q THEN 
				iStateModbusError := 300;	 
			END_IF
	
END_CASE

(*------------------------------------------------------------------Error and Warning----------------------------------------------------------------------------*)	
 
IF dwChargingState = 4 OR dwErrorCode <> 0 THEN bErrorCS := TRUE; ELSE bErrorCS := FALSE; END_IF

IF timDissableFunctions.Q THEN fbCS.bWarning := TRUE; fbCS.iWarningCode := 0; ELSE fbCS.bWarning := FALSE; END_IF   
	IF Lynus_Standards.GVL_Energy.stNumberOfDevices.diNumberOfECS > Constants_Energy.diMaxNumberOfElectricChargingStations OR bErrorCS OR byMBTCPErrorCounter > 10 THEN 
		fbCS.bError := TRUE;
	ELSE 
		fbCS.bError := FALSE;
			fbCS.iErrorCode := 0;
	END_IF

IF Lynus_Standards.GVL_Energy.stNumberOfDevices.diNumberOfECS > Constants_Energy.diMaxNumberOfElectricChargingStations THEN fbCS.iErrorCode := 1;
ELSIF bErrorCS OR byMBTCPErrorCounter > 10 THEN fbCS.iErrorCode := 0; END_IF

(*------------------------------------------------------------------Logic----------------------------------------------------------------------------*)

//Calcualte the total SOC if we have more then 1 battery in our system
diNumberOfActiveBatterys := 0;
	dwSumSOC := 0;
		FOR liLPBatteryData := 1 TO Constants_Energy.diMaxNumberOfBatterys BY 1 DO
			IF Lynus_Standards.GVL_Energy.stDataOfBatterys[diNrOfEMS_IN,liLPBatteryData].bEnabled THEN diNumberOfActiveBatterys := diNumberOfActiveBatterys + 1; END_IF
				dwSumSOC := dwSumSOC + Lynus_Standards.GVL_Energy.stDataOfBatterys[diNrOfEMS_IN,liLPBatteryData].dwSOC;
		END_FOR
	
IF diNumberOfActiveBatterys > 0 THEN
	fbCS.dwBatterySOC := DINT_TO_DWORD(DWORD_TO_DINT(dwSumSOC) / diNumberOfActiveBatterys);
ELSE
	fbCS.dwBatterySOC := 100;	//When we have no battery in the ems system
END_IF

//Check if one or more Batterysystems or batteryinverter make island mode
diNumberOfBatteryInverterInEPO := 0;
	FOR liLPInEPO := 1 TO Constants_Energy.diMaxNumberOfBatteryInverters BY 1 DO
		IF Lynus_Standards.GVL_Energy.stDataOfBatteryInverters[diNrOfEMS_IN,liLPInEPO].bWorkOnIslandMode THEN fbCS.bEPOIsActive := TRUE; diNumberOfBatteryInverterInEPO := diNumberOfBatteryInverterInEPO + 1; END_IF
	END_FOR 
		IF diNumberOfBatteryInverterInEPO <= 0 THEN fbCS.bEPOIsActive := FALSE; END_IF

//Digital input for external lock signal
fbDIExternalLock(bInvers:= FALSE, bSignal=> );

//Car connected to the ECS
IF dwCableState = 5 OR dwCableState = 7 THEN fbCS.bCarConnected := TRUE; ELSE fbCS.bCarConnected := FALSE; END_IF

//Charging time
IF dwChargingState = 3 OR dwCableState = 7 THEN timChTimeSocket.IN := TRUE; ELSE timChTimeSocket.IN := FALSE; END_IF

IF timChTimeSocket.IN THEN fbCS.arrSocketChargingTimeInput[1] := TIME_TO_REAL(timChTimeSocket.ET) / 60000; END_IF
fbCS.arrSocketChargingTimeInput[2] := 0;
fbCS.arrSocketChargingTimeInput[3] := 0;
fbCS.arrSocketChargingTimeInput[4] := 0;

timChTimeSocket(IN:= , PT:= T#24H, Q=> , ET=> );

//Mode 3 State
//Default set to No Informantion
fbCS.arrSocketMode3StateECS[1] := '';
	//Ready or Free
	IF dwChargingState = 2 THEN fbCS.arrSocketMode3StateECS[1] := 'A'; END_IF
	//Car Connected
	IF dwCableState = 5 OR dwCableState = 7 THEN fbCS.arrSocketMode3StateECS[1] := 'B1'; END_IF
	//Charging
	IF dwChargingState = 3 OR dwCableState = 7 THEN fbCS.arrSocketMode3StateECS[1] := 'C2'; END_IF
	//Error
	IF dwChargingState = 4 OR dwErrorCode <> 0 THEN fbCS.arrSocketMode3StateECS[1] := 'F'; END_IF 

fbCS.arrSocketMode3StateECS[2] := '';
fbCS.arrSocketMode3StateECS[3] := '';
fbCS.arrSocketMode3StateECS[4] := '';

//SOC Car
fbCS.arrSOCCar[1] := 0;
fbCS.arrSOCCar[2] := 0;
fbCS.arrSOCCar[3] := 0;
fbCS.arrSOCCar[4] := 0;

//Functionblock ECS
fbCS(
	bEnable:= bEnable AND NOT timDissableFunctions.Q, 
	bError:= ,
	bWarning := ,
	bEPOIsActive:= , 
	bExternalLock:= fbDIExternalLock.bSignal, 
	bCarConnected:= , 
	bWriteWithDelay:= TRUE, 
	bCalculateEnergySession:= ,
	iErrorCode:= , 
	iWarningCode:= , 
	arrSocketChargingTimeInput:= ,
	arrSOCCar:= , 
	dwBatterySOC:= , 
	lrTotalCounterEnergy_Consumption:= , 
	lrTotalCounterEnergy_Production:= , 
	lrCounterEnergyT1_Consumption:= , 
	lrCounterEnergyT2_Consumption:= , 
	lrCounterEnergyT1_Production:= , 
	lrCounterEnergyT2_Production:= , 
	lrTotalPowerECS:= , 
	arrSocketEnergySession:= ,
	rTargetPower:= Lynus_Standards.GVL_Energy.stDataElectricChargingStations[diNrOfEMS_IN,diNrOfECS_OUT].rTargetPowerEMS, 
	rSupplyVoltage:= 692, 
	rMinCurrent:= 6, 
	tTimDelayOutput:= T#5S, 
	tDelayError:= T#5S,
	arrSocketMode3StateECS:= ,
	arrSocketPowerECS:= ,
	stSetupECS:= stSetupECS, 
	stDataECSOut=> , 
	stDataECSOutDelay=> stDataECS);

//Real time Power for Output
lrTotalPowerECSRealTime := fbCS.stDataECSOut.lrTotalPower;
	
(*------------------------------------------------------------------------------------------State Machine Write---------------------------------------------------------------------------------------------*)	

CASE iStateModbusWrite OF	

	1://Set the charging current (Reg 5004)
		iStateModbus_CP := iStateModbusWrite;
		
			fbMBWrite_FC6.nMBAddr := 5004;
				fbMBWrite_FC6.bExecute := TRUE;
					fbMBWrite_FC6.nUnitID := 255;
						//Charge Current in mA
						fbMBWrite_FC6.nValue := REAL_TO_WORD(fbCS.stDataECSOut.rTargetChargeCurrent * 1000);
		
		IF fbMBWrite_FC6.bBusy THEN timDelay.IN := TRUE; END_IF

		//Wait for Delay and then next step
		IF NOT fbMBWrite_FC6.bBusy AND NOT fbMBWrite_FC6.bError AND timDelay.Q THEN
			fbMBWrite_FC6.bExecute := FALSE;
				timDelay.IN := FALSE;
					//Go to Next Step
					iStateModbusWrite := 2;
		END_IF
				
		//Error or Timout
		IF FPError_FC_6.Q OR timTimeout.Q THEN
			iStateModbusError := 300;
		END_IF
	
	2://Enable/Dissable Charging station (Reg 5014)
		iStateModbus_CP := iStateModbusWrite;
		
			fbMBWrite_FC6.nMBAddr := 5014;
				fbMBWrite_FC6.bExecute := TRUE;
					fbMBWrite_FC6.nUnitID := 255;
						//Enable and Dissable the Charging station
						IF fbCS.stDataECSOut.rTargetChargeCurrent <> 0 THEN 
							//Enable
							fbMBWrite_FC6.nValue := 1;
						ELSE
							//Dissable
							fbMBWrite_FC6.nValue := 0;
						END_IF
		
		IF fbMBWrite_FC6.bBusy THEN timDelay.IN := TRUE; END_IF

		//Wait for Delay and then next step
		IF NOT fbMBWrite_FC6.bBusy AND NOT fbMBWrite_FC6.bError AND timDelay.Q THEN
			fbMBWrite_FC6.bExecute := FALSE;
				timDelay.IN := FALSE;
					//Go to Next Step
					iStateModbusWrite := 4; // was 3/ just for testing
		END_IF
				
		//Error or Timout
		IF FPError_FC_6.Q OR timTimeout.Q THEN
			iStateModbusError := 300;
		END_IF
		
	3://Failsafe current (Reg 5016)
		iStateModbus_CP := iStateModbusWrite;
		
			fbMBWrite_FC6.nMBAddr := 5016;
				fbMBWrite_FC6.bExecute := TRUE;
					fbMBWrite_FC6.nUnitID := 255;
						//Failsafe current in mA
						fbMBWrite_FC6.nValue := uiFailsafeCurrent;
	
		IF fbMBWrite_FC6.bBusy THEN timDelay.IN := TRUE; END_IF

		//Wait for Delay and then next step
		IF NOT fbMBWrite_FC6.bBusy AND NOT fbMBWrite_FC6.bError AND timDelay.Q THEN
			fbMBWrite_FC6.bExecute := FALSE;
				timDelay.IN := FALSE;
					//Go to Next Step
					iStateModbusWrite := 4;
		END_IF
				
		//Error or Timout
		IF FPError_FC_6.Q OR timTimeout.Q THEN
			iStateModbusError := 300;
		END_IF	
		
	4://Failsafe Timeout (Reg 5018)
		iStateModbus_CP := iStateModbusWrite;
		
			fbMBWrite_FC6.nMBAddr := 5018;
				fbMBWrite_FC6.bExecute := TRUE;
					fbMBWrite_FC6.nUnitID := 255;
						//Failsafe Timeout in sec.
						fbMBWrite_FC6.nValue := uiFailsafeTimeOut;
	
		IF fbMBWrite_FC6.bBusy THEN timDelay.IN := TRUE; END_IF

		//Wait for Delay and then next step
		IF NOT fbMBWrite_FC6.bBusy AND NOT fbMBWrite_FC6.bError AND timDelay.Q THEN
			fbMBWrite_FC6.bExecute := FALSE;
				timDelay.IN := FALSE;
					byMBTCPErrorCounter := 0; 
						//Restart from new with the Read out part
						iStateModbusRead := 1;
							iStateModbusWrite := 0;
		END_IF
				
		//Error or Timout
		IF FPError_FC_6.Q OR timTimeout.Q THEN
			iStateModbusError := 300;
		END_IF	
		
END_CASE	
	
(*------------------------------------------------------------------------------------------State Machine Error---------------------------------------------------------------------------------------------*)	

CASE iStateModbusError OF
	
	300://Error
		iStateModbus_CP := iStateModbusError;
			timDelay.IN := FALSE;
				fbMBRead_FC3.bExecute := FALSE;
					fbMBWrite_FC6.bExecute := FALSE;
						byMBTCPErrorCounter := byMBTCPErrorCounter + 1;
							byMBTCPErrorCounter := LIMIT(0,byMBTCPErrorCounter,11); 		
								//Restart from new with the Read out part after an Error
								IF byMBTCPErrorCounter < 10 THEN
									iStateModbusRead := 1;	
										iStateModbusError := 0;
											iStateModbusWrite := 0;
								ELSE
									//Wait here in the Error State for the Delay Timer and then we dont have a Timeout Error
									iStateModbusRead := -1;   // was -1
										iStateModbusWrite := - 1;
											//Start from New when the Delay is paste
											IF timCloseSocket.Q THEN
												iStateModbusRead := 1;	
													iStateModbusError := 0;
														iStateModbusWrite := 0;	
															byMBTCPErrorCounter := 0;
											END_IF
								END_IF
						
END_CASE

//Timer to close the Socket after to much TCP Errors and reopen a new one
timCloseSocket(IN:= byMBTCPErrorCounter > 10 AND fbCS.stDataECSOut.bEnabled, PT:= T#1S, Q=> , ET=> );
// was t#1m
(*------------------------------------------------------------------------------------------Modbus TCP Functions---------------------------------------------------------------------------------------------*)

fbMBRead_FC3(sIPAddr:= sIPAdress, nTCPPort:= 502,cbLength:= SIZEOF(arrBuffer_FC3), pDestAddr:= ADR(arrBuffer_FC3), tTimeout:= T#5S );
	FPError_FC_3(CLK:= fbMBRead_FC3.bError, Q=> );		

fbMBWrite_FC6(sIPAddr:= sIPAdress, nTCPPort:= 502, tTimeout:= T#5S);	
	FPError_FC_6(CLK:= fbMBWrite_FC6.bError, Q=> );

(*-----------------------------------------------------------Handle data to Global structure for electric charging stations-----------------------------------------------------------------*)

//Delte al old Data on GVL after a online change or change on the variable diNrOfEMS_IDOD
IF diNrOfEMS_IN <> diNrOfEMS_IN_CP AND iStateGVLData = 0 THEN iStateGVLData := 10; END_IF 

CASE iStateGVLData OF
	
	0://Init Step
		byWaitInStep := 0;
			diCounterForGVL := 1;
	
	1://Wait for 4 Steps before clean al Data on GVL
		byWaitInStep := byWaitInStep + 1;
			IF byWaitInStep >= 4 AND fbNumberDevice.bNumberIsCalculatet THEN iStateGVLData := 2; END_IF
				//To much Devices, back to the Init step
				IF byWaitInStep >= 4 AND NOT fbNumberDevice.bNumberIsCalculatet THEN iStateGVLData := 0; END_IF	
			
	2://Clear all Data in GVL
		FOR diLPForGVL := 1 TO Constants_Energy.diMaxNumberOfEMS BY 1 DO 
			Lynus_Standards.GVL_Energy.stDataElectricChargingStations[diLPForGVL,diCounterForGVL].bEnabled := FALSE;
				Lynus_Standards.GVL_Energy.stDataElectricChargingStations[diLPForGVL,diCounterForGVL].bIsControllable := FALSE;
					Lynus_Standards.GVL_Energy.stDataElectricChargingStations[diLPForGVL,diCounterForGVL].byErrorWarning := 0;
						Lynus_Standards.GVL_Energy.stDataElectricChargingStations[diLPForGVL,diCounterForGVL].byPriority := 0;
							Lynus_Standards.GVL_Energy.stDataElectricChargingStations[diLPForGVL,diCounterForGVL].lrPower := 0;
								Lynus_Standards.GVL_Energy.stDataElectricChargingStations[diLPForGVL,diCounterForGVL].lrPowerConsumption := 0;
									Lynus_Standards.GVL_Energy.stDataElectricChargingStations[diLPForGVL,diCounterForGVL].lrPowerProduction := 0;
										Lynus_Standards.GVL_Energy.stDataElectricChargingStations[diLPForGVL,diCounterForGVL].rMaxPower := 0;
											Lynus_Standards.GVL_Energy.stDataElectricChargingStations[diLPForGVL,diCounterForGVL].byElectricFuseLine := 0;
												//Set also the target value from ems back here to 0 and not in EMS function because EMS is in Standy when we have a online change (Problem when we delete a ems function and make a online change)
												Lynus_Standards.GVL_Energy.stDataElectricChargingStations[diLPForGVL,diCounterForGVL].rTargetPowerEMS := 0;	
		END_FOR
		
			//Counter for ECS
			diCounterForGVL := diCounterForGVL + 1;
				diCounterForGVL := LIMIT(0,diCounterForGVL,Constants_Energy.diMaxNumberOfElectricChargingStations);
					//Back to the init step
					IF diCounterForGVL >= Constants_Energy.diMaxNumberOfElectricChargingStations THEN iStateGVLData := 0; END_IF

	10://Clear old Data on GVL 		
		Lynus_Standards.GVL_Energy.stDataElectricChargingStations[diNrOfEMS_IN_CP,diNrOfECS_OUT].bEnabled := FALSE;
			Lynus_Standards.GVL_Energy.stDataElectricChargingStations[diNrOfEMS_IN_CP,diNrOfECS_OUT].bIsControllable := FALSE;
				Lynus_Standards.GVL_Energy.stDataElectricChargingStations[diNrOfEMS_IN_CP,diNrOfECS_OUT].byErrorWarning := 0;
					Lynus_Standards.GVL_Energy.stDataElectricChargingStations[diNrOfEMS_IN_CP,diNrOfECS_OUT].byPriority := 0;
						Lynus_Standards.GVL_Energy.stDataElectricChargingStations[diNrOfEMS_IN_CP,diNrOfECS_OUT].lrPower := 0;
							Lynus_Standards.GVL_Energy.stDataElectricChargingStations[diNrOfEMS_IN_CP,diNrOfECS_OUT].lrPowerConsumption := 0;
								Lynus_Standards.GVL_Energy.stDataElectricChargingStations[diNrOfEMS_IN_CP,diNrOfECS_OUT].lrPowerProduction := 0;
									Lynus_Standards.GVL_Energy.stDataElectricChargingStations[diNrOfEMS_IN_CP,diNrOfECS_OUT].rMaxPower := 0;
										Lynus_Standards.GVL_Energy.stDataElectricChargingStations[diNrOfEMS_IN_CP,diNrOfECS_OUT].byElectricFuseLine := 0;
									
		diNrOfEMS_IN_CP := diNrOfEMS_IN;
			//Back to the init step
			iStateGVLData := 0;

END_CASE 	 

IF diNrOfECS_OUT > 0 AND fbNumberDevice.bNumberIsCalculatet AND diNrOfEMS_IN > 0 THEN
	Lynus_Standards.GVL_Energy.stDataElectricChargingStations[diNrOfEMS_IN,diNrOfECS_OUT].bEnabled := fbCS.stDataECSOut.bEnabled;
		Lynus_Standards.GVL_Energy.stDataElectricChargingStations[diNrOfEMS_IN,diNrOfECS_OUT].bIsControllable := TRUE;
			Lynus_Standards.GVL_Energy.stDataElectricChargingStations[diNrOfEMS_IN,diNrOfECS_OUT].byErrorWarning := fbCS.stDataECSOut.byErrorWarning;
				Lynus_Standards.GVL_Energy.stDataElectricChargingStations[diNrOfEMS_IN,diNrOfECS_OUT].byPriority := fbCS.stDataECSOut.byPriority;
					Lynus_Standards.GVL_Energy.stDataElectricChargingStations[diNrOfEMS_IN,diNrOfECS_OUT].lrPower := fbCS.stDataECSOut.lrTotalPower;
						Lynus_Standards.GVL_Energy.stDataElectricChargingStations[diNrOfEMS_IN,diNrOfECS_OUT].lrPowerConsumption := fbCS.stDataECSOut.lrTotalPowerConsumption;
							Lynus_Standards.GVL_Energy.stDataElectricChargingStations[diNrOfEMS_IN,diNrOfECS_OUT].lrPowerProduction := fbCS.stDataECSOut.lrTotalPowerProduction;
								Lynus_Standards.GVL_Energy.stDataElectricChargingStations[diNrOfEMS_IN,diNrOfECS_OUT].rMaxPower := fbCS.stDataECSOut.rMaxPower;	
									Lynus_Standards.GVL_Energy.stDataElectricChargingStations[diNrOfEMS_IN,diNrOfECS_OUT].byElectricFuseLine := byElectricFuseLine;
END_IF 

(*----------------------------------------------------------Save persistent data----------------------------------------------------------------*)

arrPD[1](lrValue:= BOOL_TO_LREAL(bEnable), bEventBasedActive=> );
arrPD[2](lrValue:= BOOL_TO_LREAL(bPowerDataInvers), bEventBasedActive=> );
arrPD[3](lrValue:= DINT_TO_LREAL(diNrOfEMS_IN), bEventBasedActive=> );
arrPD[4](lrValue:= DINT_TO_LREAL(diNrOfEM_IN_CS), bEventBasedActive=> );
arrPD[5](lrValue:= BOOL_TO_LREAL(stSetupECS.bManualyOn), bEventBasedActive=> );
arrPD[6](lrValue:= BOOL_TO_LREAL(stSetupECS.bOnEmergPowerOff), bEventBasedActive=> );
arrPD[7](lrValue:= BYTE_TO_LREAL(stSetupECS.byCSMinPower), bEventBasedActive=> );
arrPD[8](lrValue:= BYTE_TO_LREAL(stSetupECS.byDisableSOC), bEventBasedActive=> );
arrPD[9](lrValue:= BYTE_TO_LREAL(stSetupECS.byEnableSOC), bEventBasedActive=> );
arrPD[10](lrValue:= BYTE_TO_LREAL(stSetupECS.byManualyTargetPower), bEventBasedActive=> );
arrPD[11](lrValue:= BYTE_TO_LREAL(stSetupECS.byPriority), bEventBasedActive=> );
arrPD[12](lrValue:= REAL_TO_LREAL(stSetupECS.rMaxPower), bEventBasedActive=> );
arrPD[13](lrValue:= DINT_TO_LREAL(diNrOfEMS_IN_CP), bEventBasedActive=> );
arrPD[14](lrValue:= BYTE_TO_LREAL(byElectricFuseLine), bEventBasedActive=> );
arrPD[15](lrValue:= UINT_TO_LREAL(uiFailsafeCurrent), bEventBasedActive=> );
arrPD[16](lrValue:= UINT_TO_LREAL(uiFailsafeTimeOut), bEventBasedActive=> );
fbPDString(sText:= sIPAdress, bEventBasedActive=> );

END_FUNCTION_BLOCK

// ---- POUs/prgPersistent.TcPOU
PROGRAM prgPersistent
VAR
	fbUSV		: FB_WritePersistentData_CX81xx;

	fb_Reboot		: NT_reboot;
	m_Reboot		: BOOL:=FALSE;
END_VAR

fbUSV(
	eSaveModeData:= eUSVSaveMode.eSaveWhenPowerfail, 
	bLoadPersistentDataOk=> , 
	bPowerFailDetect=> , 
	bError=> , 
	bySaveProcess=> , 
	dwStorageLast24h=> , 
	udiErrorCode=> );
	
	
		
fb_Reboot(	netid := '',
			delay := 2,
			start := m_Reboot);

IF prg_SystemTime.structSystemTime.wMinute=59 AND prg_SystemTime.structSystemTime.wSecond=59 THEN // prg_SystemTime.structSystemTime.wHour=1 AND 
	m_Reboot:=TRUE;
END_IF

END_PROGRAM

// ---- POUs/prgMain.TcPOU
PROGRAM prgMain
VAR
	ADS_1: FB_ADS_Read;
	str_ADS_real_AverageRoomTemp: STRING(40);
	real_AverageRoomTemp	: REAL;											//{#lynus.ag#()}
	ton_Read_Delay: Ton;
END_VAR

// ADS Read out every minute
ton_Read_Delay( In:=TRUE AND NOT ton_Read_Delay.Q, 
				PT:=T#1M);
		
	
// start ADS read out of PLC Object ZVG
IF ton_Read_Delay.Q THEN
	str_ADS_real_AverageRoomTemp:='prgMain.real_AverageRoomTemp';
	ADS_1(	udintWriteLength:=SIZEOF(str_ADS_real_AverageRoomTemp),
			udintReadLength:=SIZEOF(real_AverageRoomTemp),
			dwSourceAddr:=ADR(str_ADS_real_AverageRoomTemp),
			dwDestAddr:=ADR(real_AverageRoomTemp),
			strNETid:='5.109.229.195.1.1');		// AMS NetID Object ZVG
END_IF

real_AverageRoomTemp := INT_TO_REAL(REAL_TO_INT(real_AverageRoomTemp*1000))/1000;

END_PROGRAM

// ---- FB/FB_ADS_Read.TcPOU
FUNCTION_BLOCK FB_ADS_Read
VAR
	intState: INT;
	fbADSRDWRT: ADSRDWRT;
	Timer1: TON;
END_VAR
VAR_INPUT
	udintWriteLength:UDINT;
	udintReadLength:UDINT;
	dwSourceAddr:pvoid;
	dwDestAddr:PVOID;
	strNetID: STRING;
END_VAR
VAR_OUTPUT
	mADSError: BOOL;
	strADSErrorText: STRING;
END_VAR

CASE intState OF
0:	(* start reading *)
	fbADSRDWRT.WRITELEN:=udintWriteLength;
	fbADSRDWRT.READLEN:=udintReadLength;
	fbADSRDWRT.SRCADDR:=dwSourceAddr;
	fbADSRDWRT.DESTADDR:=dwDestAddr;
	fbADSRDWRT.WRTRD:=TRUE;
	intState:=1000;
1000: (* wait for reply *)
	IF NOT fbADSRDWRT.BUSY THEN
		fbADSRDWRT.WRTRD:=FALSE;
		IF NOT fbADSRDWRT.ERR THEN
			strADSErrorText:='no error';
			mADSError:=FALSE;
			intState:=0;
		ELSE
			strADSErrorText:=F_AdsErrorText(fbADSRDWRT.ERRID);
			mADSError:=TRUE;
			Timer1.IN:=TRUE;
			intState:=1100;
		END_IF
	END_IF
1100: (* wait to hold state *)
	IF Timer1.Q THEN
		Timer1.IN:=FALSE;
		intState:=0;
	END_IF
ELSE
	intState:=0;
END_CASE
Timer1(PT:=t#5s);


fbADSRDWRT(
	NETID:=strNetID,
	PORT:=851,
	IDXGRP:=16#F004,
	IDXOFFS:=0,
	TMOUT:=t#10s);


(*
VAR_INPUT
        NETID           : T_AmsNetId;
        PORT            : T_AmsPort;
        IDXGRP          : UDINT;
        IDXOFFS         : UDINT;
        WRITELEN                : UDINT;
        READLEN         : UDINT;
        SRCADDR                 : DWORD;
        DESTADDR                : DWORD;
        WRTRD           : BOOL;
        TMOUT           : TIME;
END_VAR
VAR_OUTPUT
        BUSY            : BOOL;
        ERR             : BOOL;
        ERRID           : UDINT;
END_VAR

*)

END_FUNCTION_BLOCK

// ---- FB/F_AdsErrorText.TcPOU
FUNCTION F_AdsErrorText : STRING
VAR_INPUT
	nAdsError:UDINT;
END_VAR
VAR
	sText:STRING(255);
END_VAR

(*
ADS Return Codes

Fehlernummern: 0x000..., 0x500..., 0x700..., 0x1000..., 0x274C...

Global Error Codes

Hex Dez Beschreibung 
0x0 0 kein Fehler 
0x1 1 Internal error 
0x2 2 No Rtime 
0x3 3 Allocation locked memory error 
0x4 4 Insert mailbox error 
0x5 5 Wrong receive HMSG 
0x6 6 target port not found 
0x7 7 target machine not found 
0x8 8 Unknown command ID 
0x9 9 Bad task ID 
0xA 10 No IO 
0xB 11 Unknown AMS command 
0xC 12 Win 32 error 
0xD 13 Port not connected 
0xE 14 Invalid AMS length 
0xF 15 Invalid AMS Net ID 
0x10 16 Low Installation level 
0x11 17 No debug available 
0x12 18 Port disabled 
0x13 19 Port already connected 
0x14 20 AMS Sync Win32 error 
0x15 21 AMS Sync Timeout 
0x16 22 AMS Sync AMS error 
0x17 23 AMS Sync no index map 
0x18 24 Invalid AMS port 
0x19 25 No memory 
0x1A 26 TCP send error 
0x1B 27 Host unreachable 

 

Router Error Codes

Hex Dez Fehlertyp Beschreibung 
0x500 1280 Intern ROUTERERR_NOLOCKEDMEMORY
Es konnte kein nicht auslagerbarer Speicher alloziert werden. 
0x501  1281  Intern  ROUTERERR_RESIZEMEMORY
Der Routerspeicher konnte nicht in seiner Größe verändert werden.  
0x502  1282  Intern  ROUTERERR_MAILBOXFULL
Die Mailbox eines AmsPorts hat die maximal mögliche Anzahl Einträge erreicht.
Die aktuell gesendete Nachricht wurde verworfen.  
0x503  1283  Intern  ROUTERERR_DEBUGBOXFULL
Die Mailbox des Ams Debugger Ports  hat die maximal mögliche Anzahl Einträge erreicht.
Die gesendete Nachricht wird nicht im Debug Monitor angezeigt.  
0x504  1284  Intern  ROUTERERR_UNKNOWNPORTTYPE   
0x505  1285  Intern  ROUTERERR_NOTINITIALIZED
Router ist (noch) nicht initialisiert.  
0x506  1286  Intern  ROUTERERR_PORTALREADYINUSE 
Die gewünschte Portnummer ist schon vergeben.  
0x507  1287  Intern  ROUTERERR_NOTREGISTERED 
Ams Port ist nicht registriert.  
0x508  1288  Intern  ROUTERERR_NOMOREQUEUES
Die maximale Anzahl möglicher Ams Ports ist erreicht.  
0x509  1289  Intern  ROUTERERR_INVALIDPORT   
0x50A  1290  Intern  ROUTERERR_NOTACTIVATED 
Der TwinCAT Router ist (noch) nicht aktiv.  

 

General ADS Error Codes

Hex Dez Beschreibung 
0x700 1792 error class <device error> 
0x701 1793 Service is not supported by server 
0x702 1794 invalid index group 
0x703 1795 invalid index offset 
0x704 1796 reading/writing not permitted 
0x705 1797  parameter size not correct 
0x706 1798 invalid parameter value(s) 
0x707 1799 device is not in a ready state 
0x708 1800 device is busy 
0x709 1801 invalid context (must be in Windows) 
0x70A 1802 out of memory 
0x70B 1803 invalid parameter value(s) 
0x70C 1804 not found (files, ...) 
0x70D 1805 syntax error in command or file 
0x70E 1806 objects do not match 
0x70F 1807 object already exists 
0x710 1808 symbol not found 
0x711 1809 symbol version invalid 
0x712 1810 server is in invalid state 
0x713 1811 AdsTransMode not supported 
0x714 1812 Notification handle is invalid 
0x715 1813 Notification client not registered 
0x716 1814 no more notification handles 
0x717 1815 size for watch too big 
0x718 1816 device not initialized 
0x719 1817 device has a timeout 
0x71A 1818 query interface failed 
0x71B 1819 wrong interface required 
0x71C 1820 class ID is invalid 
0x71D 1821 object ID is invalid 
0x71E 1822 request is pending 
0x71F 1823 request is aborted 
0x720 1824 signal warning 
0x721 1825 invalid array index 
0x722 1826 symbol not active -> release handle and try again 
0x723 1827 access denied 
0x740 1856 Error class <client error> 
0x741 1857 invalid parameter at service 
0x742 1858 polling list is empty 
0x743 1859 var connection already in use 
0x744 1860 invoke ID in use 
0x745 1861 timeout elapsed 
0x746 1862 error in win32 subsystem 
0x748 1864 ads port not opened 
0x750 1872 internal error in ads sync 
0x751 1873 hash table overflow 
0x752 1874 key not found in hash 
0x753 1875 no more symbols in cache 
0x754 1876 invalid response received 
0x755 1877 Sync port locked
ADS-Client tries to send a ADS msg but another thread is still waiting for an ADS-response. 
This error occurs only if no ADS-router is installed (please install royalty free TwinCAT-CP) 
or the router does not know the remote ADS device (define the remote ADS partner ) 

 

RTime Error Codes

Hex Dez Fehlertyp Beschreibung 
0x1000  4096  Intern  RTERR_INTERNAL 
Interner fataler Fehler im TwinCAT Echtzeitsystem  
0x1001  4097  Intern  RTERR_BADTIMERPERIODS
Ungültiger Timerwert.  
0x1002  4098  Intern  RTERR_INVALIDTASKPTR
Task Pointer hat den ungültigen Wert NULL.  
0x1003  4099  Intern  RTERR_INVALIDSTACKPTR
Task Stack Pointer hat den ungültigen Wert NULL.  
0x1004  4100  Intern  RTERR_PRIOEXISTS
Die geforderte Taskpriorität ist schon vergeben.  
0x1005  4101  Intern  RTERR_NOMORETCB
Kein freier TCB (Task Control Block) mehr verfügbar. Maximale Anzahl von TCBs ist 64.  
0x1006  4102  Intern  RTERR_NOMORESEMAS
Keine freie Semaphore mehr verfügbar. Maximale Anzahl von Semaphoren ist 64.  
0x1007  4103  Intern  RTERR_NOMOREQUEUES
Keine freie Queue mehr verfügbar. Maximale Anzahl von Queues ist 64.  
0x1008  4104  Intern  TwinCAT reserved.  
0x1009  4105  Intern  TwinCAT reserved.  
0x100A  4106  Intern  TwinCAT reserved.  
0x100B  4107  Intern  TwinCAT reserved.  
0x100C 4108  Intern  TwinCAT reserved.  
0x100D 4109  Intern  RTERR_EXTIRQALREADYDEF
Ein externer Synchronisierungsinterrupt ist schon angemeldet.  
0x100E 4110  Intern  RTERR_EXTIRQNOTDEF
Kein externer Synchronisierungsinterrupt angemeldet.  
0x100F 4111  Intern  RTERR_EXTIRQINSTALLFAILED
Anmelden des externen Synchronisierungsinterrupts ist fehlgeschlagen.  
0x1010  4112  Intern  RTERR_IRQLNOTLESSOREQUAL
Aufruf einer Dienstfunktion im falschen Kontext.  

 

Socket Error Codes

Hex Dez Beschreibung 
0x274c 10060 A socket operation was attempted to an unreachable host 
0x274d 10061 A connection attempt failed because the connected party did not properly respond after a period of time, 
or established connection failed because connected host has failed to respond. 
0x2751 10065 No connection could be made because the target machine actively refused it 
    Weitere Socket Fehler-Codes finden Sie hier: Win32 Error Codes 

*)

CASE nAdsError OF
	0	:		sText := 'kein Fehler';
	1	:		sText := 'Internal error';
	2	:		sText := 'No Rtime';
	3	:		sText := 'Allocation locked memory error';
	4	:		sText := 'Insert mailbox error';
	5	:		sText := 'Wrong receive HMSG';
	6	:		sText := 'target port not found';
	7	:		sText := 'target machine not found';
	8	:		sText := 'Unknown command ID';
	9	:		sText := 'Bad task ID';
	10	:		sText := 'No IO';
	11	:		sText := 'Unknown AMS command';
	12	:		sText := 'Win 32 error';
	13	:		sText := 'Port not connected';
	14	:		sText := 'Invalid AMS length';
	15	:		sText := 'Invalid AMS Net ID';
	16	:		sText := 'Low Installation level';
	17	:		sText := 'No debug available';
	18	:		sText := 'Port disabled';
	19	:		sText := 'Port already connected';
	20	:		sText := 'AMS Sync Win32 error';
	21	:		sText := 'AMS Sync Timeout';
	22	:		sText := 'AMS Sync AMS error';
	23	:		sText := 'AMS Sync no index map';
	24	:		sText := 'Invalid AMS port';
	25	:		sText := 'No memory ';
	26	:		sText := 'TCP send error ';
	27	:		sText := 'Host unreachable';
	1280	:		sText := 'Router: no locked memory ';
	1282	:		sText := 'Router: mailbox full ';
	1792	:		sText := 'error class <device error> ';
	1793	:		sText := 'Service is not supported by server ';
	1794	:		sText := 'invalid index group ';
	1795	:		sText := 'invalid index offset ';
	1796	:		sText := 'reading-writing not permitted ';
	1797	:		sText:='parameter size not correct';
	1798	:		sText := 'invalid parameter value ';
	1799	:		sText := 'device is not in a ready state ';
	1800	:		sText := 'device is busy ';
	1801	:		sText := 'invalid context (must be in Windows) ';
	1802	:		sText := 'out of memory';
	1803	:		sText := 'invalid parameter value(s)';
	1804	:		sText := 'not found (files, ...)';
	1805	:		sText := 'syntax error in command or file';
	1806	:		sText := 'objects do not match';
	1807	:		sText := 'object already exists';
	1808	:		sText := 'symbol not found';
	1809	:		sText := 'symbol version invalid';
	1810	:		sText := 'server is in invalid state';
	1811	:		sText := 'AdsTransMode not supported';
	1812	:		sText := 'Notification handle is invalid';
	1813	:		sText := 'Notification client not registered';
	1814	:		sText := 'no more notification handles';
	1815	:		sText := 'size for watch too big';
	1816	:		sText := 'device not initialized';
	1817	:		sText := 'device has a timeout';
	1818	:		sText := 'query interface failed';
	1819	:		sText := 'wrong interface required';
	1820	:		sText := 'class ID is invalid';
	1821	:		sText := 'object ID is invalid';
	1822	:		sText := 'request is pending';
	1823	:		sText := 'request is aborted';
	1824	:		sText := 'signal warning';
	1825	:		sText := 'invalid array index';
	1856	:		sText := 'Error class <client error>';
	1857	:		sText := 'invalid parameter at service';
	1858	:		sText := 'polling list is empty';
	1859	:		sText := 'var connection already in use';
	1860	:		sText := 'invoke ID in use';
	1861	:		sText := 'timeout elapsed';
	1862	:		sText := 'error in win32 subsystem';
	1864	:		sText := 'ads port not opened';
	1872	:		sText := 'internal error in ads sync';
	1873	:		sText := 'hash table overflow';
	1874	:		sText := 'key not found in hash';
	1875	:		sText := 'no more symbols in cache';
	1877	:		sText := 'Sync port locked: ADS-Client tries to send a ADS msg but another thread is still waiting for an ADS-response. This error occurs only if no ADS-router is installed or the router does not know the remote ADS device (define the remote ADS partner )';
	10060	:		sText := 'A socket operation was attempted to an unreachable host';
	10061	:		sText := 'A connection attempt failed because the connected party did not properly respond after a period of time, or established connection failed because connected host has failed to respond.';
	10065	:		sText := 'No connection could be made because the target machine actively refused it';

(* FB_SmtpV2 *)
	32778 	:	sText := 'Not connected';
	32779 	:	sText := 'Sender expected';
	32780 	:	sText := 'Recipients expected';
	32781 	:	sText := 'Send FROM command failed';
	32782 	:	sText := 'Send DATA command failed';
	32783 	:	sText := 'Send mail header failed';
	32784 	:	sText := 'Send mail body failed';
	32785 	:	sText := 'Send "end of mail indicator" failed';
	32786 	:	sText := 'Send "RCPT" command failed';
	32787 	:	sText := 'Server Response got no username request';
	32788 	:	sText := 'Server Response got no password request';
	32789 	:	sText := 'Unable to create socket connection';
	32790 	:	sText := 'Authentication type not supported by smtp server';
	32791 	:	sText := 'Wrong username or password';
	32792 	:	sText := 'Not supported';
	32793 	:	sText := 'Invalid hostname';
	32794 	:	sText := 'Unable to send attachment';
	32795 	:	sText := 'File not found';
	32796 	:	sText := 'Invalid Version (New SMTP Server with old SMTP PLC library)';
	32797 	:	sText := 'Unable to connect (Connection error => sometimes wrong port or wrong server)';
	32798 	:	sText := 'Unable to create socket';
	32799 	:	sText := 'WSA startup failed';
	32800 	:	sText := 'Invalid hostname';
	32801 	:	sText := 'Unecpected response from server';
	32802 	:	sText := 'Error while receiving data';
	32803 	:	sText := 'No supported authentication methods found';
	32804 	:	sText := 'Invalid parameter';
	32928 	:	sText := 'Security interface not found';
	32929 	:	sText := 'Unable to call security interface';
	32930 	:	sText := 'Security initialization failed';
	32932 	:	sText := 'Unable to create credentials';
	32933 	:	sText := 'SSL-handshake failed';
	32934 	:	sText := 'Invalid server credentials';
	32935 	:	sText := 'Unable to verify server';
	32936 	:	sText := 'Unable to encrypt message';
	32937 	:	sText := 'Unable to decrypt message';


	ELSE			sText := 'Error not defined';
END_CASE;

F_ADSerrorText := sText;

END_FUNCTION

// ---- FB/FB_Shelly_3EM_not_tested.TcPOU
FUNCTION_BLOCK FB_Shelly_3EM_not_tested
VAR_INPUT
	bStart				: BOOL;
	tDelayRequest		: TIME;		//Timer for delay before start with the next read or write Request
	sHostname			: STRING(255);		//Hostname or IP Adress from the Server
END_VAR

VAR_IN_OUT
END_VAR

VAR_OUTPUT
	bValidResult		: BOOL;							//Valid Result received from Server
    bBusy				: BOOL;							//Function is Busy
    bError				: BOOL;							//Error sucess
	bDone				: BOOL;							//True after the decoding from the received Json File
	bConnected			: BOOL;							//Connection to the Server
	lrtotalpower		: LREAL;						//Received Value
	lrpowerL1			: LREAL;
	lrcurrentL1			: LREAL;
	lrvoltageL1			: LREAL;
	lrenergyL1			: LREAL;
	lrpowerL2			: LREAL;
	lrcurrentL2			: LREAL;
	lrvoltageL2			: LREAL;
	lrenergyL2			: LREAL;
	lrpowerL3			: LREAL;
	lrcurrentL3			: LREAL;
	lrvoltageL3			: LREAL;
	lrenergyL3			: LREAL;
	hrErrorCode       	: HRESULT;						//Error Result from Http Client
END_VAR

VAR
	fbClient			: FB_IotHttpClient;
	fbHttpGet			: FB_Shelly_3EM_Helper;
	timStartRequest		: TON;							//Timer to Start the Request
	FPStartRequest		: R_TRIG;						//Internal positive Edge
	FPDone				: R_TRIG;						//Internal positive Edge
	FNStart				: F_TRIG;						//Internal negative Edge
	y: INT;
	mtest: BOOL;
END_VAR

(*------------------------------------------------------------------------------------Configure HTTP Client------------------------------------------------------------------------------------------------------*)

fbClient.sHostName := sHostname;
fbClient.tConnectionTimeout := T#30S;

IF NOT fbClient.bConfigured THEN 
	fbClient.nHostPort:= 80;
	fbClient.bKeepAlive := TRUE;
	fbClient.tConnectionTimeout := T#30S;
	fbClient.stTLS.bNoServerCertCheck := TRUE;
END_IF


//Timer to start the Request
FPStartRequest(CLK:= bStart, Q=> );
timStartRequest(IN:= fbClient.bConfigured AND bStart AND NOT timStartRequest.Q, PT:= tDelayRequest, Q=> , ET=> );

IF ((timStartRequest.Q AND NOT bBusy AND fbClient.bConnected) OR (FPStartRequest.Q AND NOT bBusy AND fbClient.bConfigured AND fbClient.bConnected)) THEN 
	y:=y+1;
	fbHttpGet.bSend := TRUE; 
END_IF

				
//Http Get Function
fbHttpGet(
	lrtotalpower => lrtotalpower, 
	lrpowerL1 => lrpowerL1,
	lrcurrentL1 => lrcurrentL1,
	lrvoltageL1 => lrvoltageL1,
	lrenergyL1 => lrenergyL1,
	lrpowerL2 => lrpowerL2,
	lrcurrentL2 => lrcurrentL2,
	lrvoltageL2 => lrvoltageL2,
	lrenergyL2 => lrenergyL2,
	lrpowerL3 => lrpowerL3,
	lrcurrentL3 => lrcurrentL3,
	lrvoltageL3 => lrvoltageL3,
	lrenergyL3 => lrenergyL3,
	bSend:= , 
	fbClient:= fbClient, 
	bBusy=> bBusy, 
	bError=> ,
	sContentStatus=> ,
	sContentM0=> ,
	sContentM1=> ,
	sContentM2=> );


fbHttpGet.bSend := FALSE;

FPDone(CLK:= bDone, Q=> );

(*
//Http Client
FNStart(CLK:= bStart, Q=> );
	IF FNStart.Q THEN fbClient.Disconnect(); END_IF
*)
IF mtest THEN
	fbClient.Disconnect();
	mtest:=FALSE;
ELSE
	fbClient.Execute();	
END_IF

//Error
IF fbHttpGet.bError OR fbClient.bError THEN 
	bError := TRUE; 
ELSE 
	bError := FALSE; 
END_IF	

hrErrorCode := fbClient.hrErrorCode;

END_FUNCTION_BLOCK

// ---- FB/FB_Shelly_3EM_Helper_not_tested.TcPOU
FUNCTION_BLOCK FB_Shelly_3EM_Helper_not_tested
VAR_INPUT
	bSend				: BOOL;
END_VAR

VAR_IN_OUT
	fbClient			: FB_IotHttpClient;
END_VAR

VAR_OUTPUT
	bBusy				: BOOL;
	bError				: BOOL;
	lrtotalpower		: LREAL;
	lrpowerL1			: LREAL;
	lrcurrentL1			: LREAL;
	lrvoltageL1			: LREAL;
	lrenergyL1			: LREAL;
	lrpowerL2			: LREAL;
	lrcurrentL2			: LREAL;
	lrvoltageL2			: LREAL;
	lrenergyL2			: LREAL;
	lrpowerL3			: LREAL;
	lrcurrentL3			: LREAL;
	lrvoltageL3			: LREAL;
	lrenergyL3			: LREAL;
END_VAR

VAR
	fbRequestStatus		: FB_IotHttpRequest;
	fbRequestMeter0		: FB_IotHttpRequest;
	fbRequestMeter1		: FB_IotHttpRequest;
	fbRequestMeter2		: FB_IotHttpRequest;
	fbJson				: FB_JsonDomParser;
	nState				: UDINT;
	RisingEdge			: R_TRIG;
	timTimeout			: TON;
	tTimeOut			: TIME := T#50S;
	bGetContentResult	: BOOL;
	sContentStatus		: STRING(511);
	sContentM0			: STRING(511);
	sContentM1			: STRING(511);
	sContentM2			: STRING(511);
	
	bGetJsonResult		: BOOL;
	jsonDoc				: SJsonValue;
	jsonVal				: SJsonValue;
	
	nReqCount			: UDINT;	
	nResCount			: UDINT;
	nValidResCount		: UDINT;
	nErrCount			: UDINT;
	x: INT;
END_VAR

//Timer for Timeout
timTimeout(IN:= nState = 1 AND bBusy, PT:= tTimeOut, Q=> , ET=> );
	IF timTimeout.Q THEN 
		nState := 0;
		bBusy := FALSE;
	END_IF

RisingEdge(CLK:= bSend );
CASE nState OF
0:	// wait for trigger
	IF RisingEdge.Q THEN 
		nState :=1;
	END_IF

1:	// first request	
	bBusy:= TRUE;
	bError:= FALSE;
	IF	fbRequestStatus.SendRequest(sUri:='/status', fbClient:=fbClient, eRequestType:=ETcIotHttpRequestType.HTTP_Get, 0, 0, 0) THEN
		nState:= 2;
		nReqCount:= nReqCount+1;
	END_IF

2:	// second request	
	IF	fbRequestMeter0.SendRequest(sUri:='/emeter/0', fbClient:=fbClient, eRequestType:=ETcIotHttpRequestType.HTTP_Get, 0, 0, 0) THEN
		nState:= 3;
		nReqCount:= nReqCount+1;
	END_IF

3:	// third request	
	IF fbRequestMeter1.SendRequest(sUri:='/emeter/1', fbClient:=fbClient, eRequestType:=ETcIotHttpRequestType.HTTP_Get, 0, 0, 0) THEN
		nState:= 4;
		nReqCount:= nReqCount+1;
	END_IF

4:	// fourth request	
	IF  fbRequestMeter2.SendRequest(sUri:='/emeter/2', fbClient:=fbClient, eRequestType:=ETcIotHttpRequestType.HTTP_Get, 0, 0, 0) THEN
		nState:= 5;
		nReqCount:= nReqCount+1;
	END_IF

5: //Convert Data
	IF NOT fbRequestMeter0.bBusy AND NOT fbRequestMeter1.bBusy AND NOT fbRequestMeter2.bBusy AND NOT fbRequestStatus.bBusy THEN
		bError:= TRUE;
		IF NOT fbRequestMeter0.bError THEN				 
			bGetContentResult:= fbRequestMeter0.GetContent(pContent:= ADR(sContentM0), nContentSize:= SIZEOF(sContentM0), bSetNullTermination:= TRUE);
			IF fbRequestMeter0.nStatusCode >= 200 AND fbRequestMeter0.nStatusCode < 300 THEN
				bGetJsonResult:= FALSE;
				jsonDoc:= fbRequestMeter0.GetJsonDomContent(fbJson);
				IF jsonDoc <> 0 THEN
					bGetJsonResult:= TRUE;
					IF fbJson.HasMember(jsonDoc, 'power')  THEN
						jsonVal:= fbJson.FindMember(jsonDoc, 'power');
						nValidResCount:= nValidResCount+1;
						IF fbJson.IsDouble(jsonVal) THEN							
							lrpowerL1:= fbJson.GetDouble(jsonVal);									
						END_IF
						jsonVal:= fbJson.FindMember(jsonDoc, 'current');
						nValidResCount:= nValidResCount+1;
						IF fbJson.IsDouble(jsonVal) THEN							
							lrcurrentL1:= fbJson.GetDouble(jsonVal);									
						END_IF
						jsonVal:= fbJson.FindMember(jsonDoc, 'voltage');
						nValidResCount:= nValidResCount+1;
						IF fbJson.IsDouble(jsonVal) THEN							
							lrvoltageL1:= fbJson.GetDouble(jsonVal);									
						END_IF
						jsonVal:= fbJson.FindMember(jsonDoc, 'total');
						nValidResCount:= nValidResCount+1;
						IF fbJson.IsDouble(jsonVal) THEN							
							lrenergyL1:= fbJson.GetDouble(jsonVal);									
						END_IF	
						bError:= FALSE;
						END_IF
					END_IF						
				nResCount:= nResCount+1;			
				END_IF
		END_IF
		
		IF NOT fbRequestMeter1.bError THEN				 
			bGetContentResult:= fbRequestMeter1.GetContent(pContent:= ADR(sContentM1), nContentSize:= SIZEOF(sContentM1), bSetNullTermination:= TRUE);
			IF fbRequestMeter1.nStatusCode >= 200 AND fbRequestMeter1.nStatusCode < 300 THEN
				bGetJsonResult:= FALSE;
				jsonDoc:= fbRequestMeter1.GetJsonDomContent(fbJson);
				IF jsonDoc <> 0 THEN
					bGetJsonResult:= TRUE;
					IF fbJson.HasMember(jsonDoc, 'power')  THEN
						jsonVal:= fbJson.FindMember(jsonDoc, 'power');
						nValidResCount:= nValidResCount+1;
						IF fbJson.IsDouble(jsonVal) THEN							
							lrpowerL2:= fbJson.GetDouble(jsonVal);									
						END_IF
						jsonVal:= fbJson.FindMember(jsonDoc, 'current');
						nValidResCount:= nValidResCount+1;
						IF fbJson.IsDouble(jsonVal) THEN							
							lrcurrentL2:= fbJson.GetDouble(jsonVal);									
						END_IF
						jsonVal:= fbJson.FindMember(jsonDoc, 'voltage');
						nValidResCount:= nValidResCount+1;
						IF fbJson.IsDouble(jsonVal) THEN							
							lrvoltageL2:= fbJson.GetDouble(jsonVal);									
						END_IF
						jsonVal:= fbJson.FindMember(jsonDoc, 'total');
						nValidResCount:= nValidResCount+1;
						IF fbJson.IsDouble(jsonVal) THEN							
							lrenergyL2:= fbJson.GetDouble(jsonVal);									
						END_IF	
						bError:= FALSE;
						END_IF
					END_IF						
				nResCount:= nResCount+1;			
				END_IF
		END_IF
		
		IF NOT fbRequestMeter2.bError THEN				 
			bGetContentResult:= fbRequestMeter2.GetContent(pContent:= ADR(sContentM2), nContentSize:= SIZEOF(sContentM2), bSetNullTermination:= TRUE);
			IF fbRequestMeter2.nStatusCode >= 200 AND fbRequestMeter2.nStatusCode < 300 THEN
				bGetJsonResult:= FALSE;
				jsonDoc:= fbRequestMeter2.GetJsonDomContent(fbJson);
				IF jsonDoc <> 0 THEN
					bGetJsonResult:= TRUE;
					IF fbJson.HasMember(jsonDoc, 'power')  THEN
						jsonVal:= fbJson.FindMember(jsonDoc, 'power');
						nValidResCount:= nValidResCount+1;
						IF fbJson.IsDouble(jsonVal) THEN							
							lrpowerL3:= fbJson.GetDouble(jsonVal);									
						END_IF
						jsonVal:= fbJson.FindMember(jsonDoc, 'current');
						nValidResCount:= nValidResCount+1;
						IF fbJson.IsDouble(jsonVal) THEN							
							lrcurrentL3:= fbJson.GetDouble(jsonVal);									
						END_IF
						jsonVal:= fbJson.FindMember(jsonDoc, 'voltage');
						nValidResCount:= nValidResCount+1;
						IF fbJson.IsDouble(jsonVal) THEN							
							lrvoltageL3:= fbJson.GetDouble(jsonVal);									
						END_IF
						jsonVal:= fbJson.FindMember(jsonDoc, 'total');
						nValidResCount:= nValidResCount+1;
						IF fbJson.IsDouble(jsonVal) THEN							
							lrenergyL3:= fbJson.GetDouble(jsonVal);									
						END_IF	
						bError:= FALSE;
						END_IF
					END_IF						
				nResCount:= nResCount+1;			
				END_IF
		END_IF
		
		IF NOT fbRequestStatus.bError THEN				 
			bGetContentResult:= fbRequestStatus.GetContent(pContent:= ADR(sContentStatus), nContentSize:= SIZEOF(sContentStatus), bSetNullTermination:= TRUE);
			IF fbRequestStatus.nStatusCode >= 200 AND fbRequestStatus.nStatusCode < 300 THEN
				bGetJsonResult:= FALSE;
				jsonDoc:= fbRequestStatus.GetJsonDomContent(fbJson);
				IF jsonDoc <> 0 THEN
					bGetJsonResult:= TRUE;
					IF fbJson.HasMember(jsonDoc, 'total_power')  THEN
						jsonVal:= fbJson.FindMember(jsonDoc, 'total_power');
						nValidResCount:= nValidResCount+1;
						IF fbJson.IsDouble(jsonVal) THEN							
							lrtotalpower:= fbJson.GetDouble(jsonVal);									
						END_IF
						bError:= FALSE;
					END_IF
				END_IF		
				nResCount:= nResCount+1;			
			END_IF
		END_IF
		
		nState:= 0;
		bBusy:= FALSE;
		IF bError THEN
			nErrCount:= nErrCount+1;
		END_IF
	END_IF  	
END_CASE

END_FUNCTION_BLOCK

// ---- POUs/prgComEffIO.TcPOU
PROGRAM prgComEffIO
VAR
	fbCom		: FB_MqttCommunicator_V2;
END_VAR

fbCom(
	bConnect:= TRUE, 
	strAuthKey:= 'BE736352867778' , 
	sUserName:= '96961966-4b77-40e7-93b8-7360bccc2c2b', 
	sUserPassword:= '6c4bf1d7-cda1-4704-a710-a6791f53ebb8' , 
	eSavePositionCertificate:= , 
	time_HeartBeat_sec:= , 
	bConnected=> , 
	bError=> , 
	hrErrorCode=> , 
	eConnectionState=> , 
	eErrorMessage_Out=> );
	
	
(* old

fbCom(
	bConnect:= TRUE, 
	sUserName:= 'a27b4241-b569-45d2-9103-231b1e1447ff', 
	sUserPassword:= '9a1076be-075f-42fd-bfbd-529176568a3e', 
	eSavePositionCertificate:= eSavePositionOnPLC.ePostionHardDisk, 
	bConnected=> , 
	bError=> , 
	hrErrorCode=> , 
	eConnectionState=> , 
	eErrorMessage_Out=> );

	*)

END_PROGRAM
